# B&R Automation Studio project 8238 (part 16)

```iecst
										_dim1 := MAX(1, _getContainerParamNum.wDimension[1]);
										_dim2 := MAX(1, _getContainerParamNum.wDimension[2]);
										_dim3 := MAX(1, _getContainerParamNum.wDimension[3]);
										_dim4 := MAX(1, _getContainerParamNum.wDimension[4]);

										FOR _i1 := _getContainerParamNum.wMinBound[1] TO _getContainerParamNum.wMinBound[1] + _dim1-1 DO

											FOR _i2 := _getContainerParamNum.wMinBound[2] TO _getContainerParamNum.wMinBound[2] + _dim2 -1 DO

												FOR _i3 := _getContainerParamNum.wMinBound[3] TO _getContainerParamNum.wMinBound[3] + _dim3 -1 DO

													FOR _i4 := _getContainerParamNum.wMinBound[4] TO _getContainerParamNum.wMinBound[4] + _dim4 -1 DO

														IF _wIdxCsvNum <= _PmIntern.CSVDataObjects.MaxIndex.lCSVNum THEN

															_pDoContainerNum.CsvNum[_wIdxCsvNum].wIdxNumPar := _i;
															_pDoContainerNum.CsvNum[_wIdxCsvNum].bRowType := _pDoParamNum.ParamNum[_i].bRowType;
															_pDoContainerNum.CsvNum[_wIdxCsvNum].diValue := _pDoParamNum.ParamNum[_i].diDefValue;

															IF _getContainerParamNum.wCountArray >= 1 THEN

																_pDoContainerNum.CsvNum[_wIdxCsvNum].wArrIdx1 := _i1;

																IF _getContainerParamNum.wCountArray >= 2 THEN

																	_pDoContainerNum.CsvNum[_wIdxCsvNum].wArrIdx2 := _i2;

																	IF _getContainerParamNum.wCountArray >= 3 THEN

																		_pDoContainerNum.CsvNum[_wIdxCsvNum].wArrIdx3 := _i3;

																		IF _getContainerParamNum.wCountArray = 4 THEN

																			_pDoContainerNum.CsvNum[_wIdxCsvNum].wArrIdx4 := _i4;

																		END_IF

																	END_IF

																END_IF

															END_IF

															_wIdxCsvNum := _wIdxCsvNum + 1;

														END_IF

													END_FOR

												END_FOR

											END_FOR

										END_FOR

									END_IF

								END_FOR

								//****************************************************************************************************************
								// Datenobjekte beschreiben (STRING)
								//****************************************************************************************************************
								_wIdxCsvString := 1;

								FOR _i := 1 TO UDINT_TO_UINT(_PmIntern.DataObjects.MaxIndex.lParamString) DO

									_getContainerParamString(enable := TRUE, pLogicStructs := ADR(_pDoLogicalStruct.LogicalStruct[1]), wMaxIdxLogicStructs := UDINT_TO_UINT(_PmIntern.DataObjects.MaxIndex.lLogicalStruct), pParamString := ADR(_pDoParamString.ParamString[_i]));

									IF _getContainerParamString.status = ERR_OK AND _getContainerParamString.iContainer = _pDoContainer.Container[_c].siContainerID THEN

										_dim1 := MAX(1, _getContainerParamString.wDimension[1]);
										_dim2 := MAX(1, _getContainerParamString.wDimension[2]);
										_dim3 := MAX(1, _getContainerParamString.wDimension[3]);
										_dim4 := MAX(1, _getContainerParamString.wDimension[4]);

										FOR _i1 := _getContainerParamString.wMinBound[1] TO _getContainerParamString.wMinBound[1] + _dim1 - 1 DO

											FOR _i2 := _getContainerParamString.wMinBound[2] TO _getContainerParamString.wMinBound[2] + _dim2 - 1 DO

												FOR _i3 := _getContainerParamString.wMinBound[3] TO _getContainerParamString.wMinBound[3] + _dim3 - 1 DO

													FOR _i4 := _getContainerParamString.wMinBound[4] TO _getContainerParamString.wMinBound[4] + _dim4 - 1 DO

														IF _wIdxCsvString <= _PmIntern.CSVDataObjects.MaxIndex.lCSVString THEN

															_pDoContainerString.CsvString[_wIdxCsvString].wIdxStringPar := _i;
															brwcsncpy(ADR(_pDoContainerString.CsvString[_wIdxCsvString].utfValue), ADR(_pDoParamString.ParamString[_i].utfDefValue), 31);

															IF _getContainerParamString.wCountArray >= 1 THEN

																_pDoContainerString.CsvString[_wIdxCsvString].wArrIdx1 := _i1;

																IF _getContainerParamString.wCountArray >= 2 THEN

																	_pDoContainerString.CsvString[_wIdxCsvString].wArrIdx2 := _i2;

																	IF _getContainerParamString.wCountArray >= 3 THEN

																		_pDoContainerString.CsvString[_wIdxCsvString].wArrIdx3 := _i3;

																		IF _getContainerParamString.wCountArray = 4 THEN

																			_pDoContainerString.CsvString[_wIdxCsvString].wArrIdx4 := _i4;

																		END_IF

																	END_IF

																END_IF

															END_IF

															_wIdxCsvString := _wIdxCsvString + 1;

														END_IF

													END_FOR

												END_FOR

											END_FOR

										END_FOR

									END_IF

								END_FOR

								//****************************************************************************************************************
								// Datenobjekte anlegen
								//****************************************************************************************************************

								_dcCSVNum(enable := TRUE, grp := 0, pName := ADR(_PmIntern.ActContainer.sDoNameNum), len := _PmIntern.CSVDataObjects.Size.lCSVNum, MemType := doUSRROM, Option := 0, pCpyData := _PmIntern.CSVDataObjects.TempAdresses.lCSVNum);

								IF (_dcCSVNum.status = ERR_OK) THEN
									_PmIntern.CSVDataObjects.Idents.lCSVNum := _dcCSVNum.ident;
									_PmIntern.CSVDataObjects.Adress.lCSVNum := _dcCSVNum.pDatObjMem;
									_PmIntern.CSVDataObjects.Size.lCSVNum := _dcCSVNum.len;

									_pDoContainerNum ACCESS _PmIntern.CSVDataObjects.Adress.lCSVNum;

									// Es muss auch eine CSV-Datei geschrieben werden
									_PmIntern.xExportContainerCsv := TRUE;

								ELSE

									_PmIntern.Logger.logLevel 	:= arlogLEVEL_INFO;
									_PmIntern.Logger.text		:= 'Create Data Object Numeric failed: Index = {##AttrVar1}. Status: {##AttrVar2}';
									_PmIntern.Logger.var1		:= _PmIntern.ActContainer.siContainerID;
									_PmIntern.Logger.var2		:= _dcCSVNum.status;
									_PmIntern.Logger();

								END_IF

								_dcCSVString(enable := TRUE, grp := 0, pName := ADR(_PmIntern.ActContainer.sDoNameString), len := _PmIntern.CSVDataObjects.Size.lCSVString, MemType := doUSRROM, Option := 0, pCpyData :=_PmIntern.CSVDataObjects.TempAdresses.lCSVString);

								IF (_dcCSVString.status = ERR_OK) THEN
									_PmIntern.CSVDataObjects.Idents.lCSVString := _dcCSVString.ident;
									_PmIntern.CSVDataObjects.Adress.lCSVString := _dcCSVString.pDatObjMem;
									_PmIntern.CSVDataObjects.Size.lCSVString := _dcCSVString.len;

									_pDoContainerString ACCESS _PmIntern.CSVDataObjects.Adress.lCSVString;

									// Es muss auch eine CSV-Datei geschrieben werden
									_PmIntern.xExportContainerCsv := TRUE;

								ELSE

									_PmIntern.Logger.logLevel 	:= arlogLEVEL_INFO;
									_PmIntern.Logger.text		:= 'Create Data Object String failed: Index = {##AttrVar1}. Status: {##AttrVar2}';
									_PmIntern.Logger.var1		:= _PmIntern.ActContainer.siContainerID;
									_PmIntern.Logger.var2		:= _dcCSVString.status;
									_PmIntern.Logger();

								END_IF

								_MemPartFree(enable := TRUE, ident := _MemPartCreate.ident, mem := _PmIntern.CSVDataObjects.TempAdresses.lCSVNum);
								_PmIntern.CSVDataObjects.TempAdresses.lCSVNum := 0;

								_MemPartFree(enable := TRUE, ident := _MemPartCreate.ident, mem := _PmIntern.CSVDataObjects.TempAdresses.lCSVString);
								_PmIntern.CSVDataObjects.TempAdresses.lCSVString := 0;

							ELSE

								_PmIntern.Logger.logLevel 	:= arlogLEVEL_INFO;
								_PmIntern.Logger.text		:= 'MemPartAlloc for Data Object String: Index = {##AttrVar1}. Status: {##AttrVar2}';
								_PmIntern.Logger.var1		:= _PmIntern.ActContainer.siContainerID;
								_PmIntern.Logger.var2		:= _MemPartAlloc.status;
								_PmIntern.Logger();

							END_IF //IF _MemPartAlloc.status = ERR_OK

						ELSE

							_PmIntern.Logger.logLevel 	:= arlogLEVEL_INFO;
							_PmIntern.Logger.text		:= 'MemPartAlloc for Data Object Numeric: Index = {##AttrVar1}. Status: {##AttrVar2}';
							_PmIntern.Logger.var1		:= _PmIntern.ActContainer.siContainerID;
							_PmIntern.Logger.var2		:= _MemPartAlloc.status;
							_PmIntern.Logger();

						END_IF

					END_IF // Direkte Parametrierung

				END_IF // Müssen Datenobjekte angelegt werden

				// Wenn SINGLEmnParam definiert ist, dann wartet die Ausführung hier solange, bis _lSingleStep > _pl_InitState gesetzt wurde
				#ifdef SINGLEmnParam
				REPEAT
		UNTIL
					(_lSingleStep > _pl_InitState) AND (_lLoop >= _lLoopCount) OR NOT _xSingleStep
				END_REPEAT
#endif

				//****************************************************************************************************************
				// CSV-Datei auf Datum prüfen und ggf. einlesen
				//****************************************************************************************************************

				_PmIntern.enInitState := is_TestFileDate;

				// Wenn Datei gefunden, dann Version und Datum bestimmen

				IF _PmIntern.Parse.lFileAdress <> 0   THEN

					brsmemset(_PmIntern.Parse.lLineTableAdress, 0, MNPARAM_MAXPARSELINES * SIZEOF(UDINT));
					brsmemset(_PmIntern.Parse.lLineTableLen, 0, MNPARAM_MAXPARSELINES * SIZEOF(UINT));

					_CountLines.enable 	:= TRUE;
					_CountLines.pFile 		:= _PmIntern.Parse.lFileAdress;
					_CountLines.FileSize 	:= _PmIntern.Parse.lFileSize;
					_CountLines.MaxLines	:= MNPARAM_MAXPARSELINES;
					_CountLines.pAdresses	:= _PmIntern.Parse.lLineTableAdress;
					_CountLines.pLens		:= _PmIntern.Parse.lLineTableLen;

					_CountLines();

					IF _CountLines.status = ERR_OK THEN

						_PmIntern.Parse.lCntLines := _CountLines.CntLines;

						// Suche Versionszeile

						_wStartLine := 1;
						_xFoundVersion := FALSE;
						_xFoundDate := FALSE;
						_xFoundMachineNo := FALSE;

						REPEAT

							_GetCsvDat.enable := TRUE;
							brwcsncpy( ADR(_GetCsvDat.utfCsvString), _plLineAdress[_wStartLine], MIN(299, _pwLineLen[_wStartLine]));
							_GetCsvDat();
							IF _GetCsvDat.RowType = MNPARAM_CSV_HEADER_VERSION THEN

								_CsvHeaderVersion := _GetCsvDat.HeaderVersion;
								_xFoundVersion := TRUE;

							ELSIF _GetCsvDat.RowType = MNPARAM_CSV_HEADER_TIMESTAMP THEN

								_CsvHeaderDate := _GetCsvDat.HeaderTime;
								_xFoundDate := TRUE;

							ELSIF _GetCsvDat.RowType = MNPARAM_CSV_HEADER_MACHINENO THEN

								_CsvHeaderMachineNo := _GetCsvDat.HeaderMachineNo;
								_xFoundMachineNo := TRUE;

							END_IF

							_wStartLine := _wStartLine + 1;

						UNTIL
							(_xFoundDate AND _xFoundVersion AND _xFoundMachineNo) OR _wStartLine > _PmIntern.Parse.lCntLines
						END_REPEAT

						_PmIntern.ActContainer.xDataImported := FALSE;

						IF _xFoundDate AND _xFoundVersion AND _xFoundMachineNo THEN

							// Ist der Maschinentyp OK ?
							IF brwcscmp(ADR(_CsvHeaderVersion.utfMachineType),ADR(_pDoContainer.Header.Version.utfMachineType)) = 0 THEN

								// Ist die Maschinennummer OK ?
								IF brwcscmp(ADR(_CsvHeaderMachineNo.utfMachineNo),ADR(IFmnParam.Out.utfMachineNumber)) = 0 THEN

									// Ist die CSV-Datei neuer als die Daten in den DO ?
									IF _pDoContainerNum.Header.Time.dtTimestamp < _CsvHeaderDate.dtTimestamp THEN

										//****************************************************************************************************************
										// Datenobjekte für das Importieren in den Hauptspeicher kopieren
										//****************************************************************************************************************

										_PmIntern.enInitState := is_ImportData1;

										//##20110901AH
										_PmIntern.Logger.logLevel 	:= arlogLEVEL_INFO;
										_PmIntern.Logger.text		:= 'Import Container Index = {##AttrVar1}. Index: {##AttrVar2}';
										_PmIntern.Logger.var1		:= _PmIntern.ActContainer.siContainerID;
										_PmIntern.Logger.var2		:= _PmIntern.ActContainer.wIndexIndirect;
										_PmIntern.Logger();

										// Numerische Daten
										_diCSVNum(enable := TRUE, pName := ADR(_PmIntern.ActContainer.sDoNameNum));

										IF _diCSVNum.status = ERR_OK THEN

											_PmIntern.CSVDataObjects.Idents.lCSVNum := _diCSVNum.ident;
											_PmIntern.CSVDataObjects.Adress.lCSVNum := _diCSVNum.pDatObjMem;
											_PmIntern.CSVDataObjects.Size.lCSVNum := _diCSVNum.len;

											_MemPartAlloc(enable :=TRUE, ident := _MemPartCreate.ident, len := _diCSVNum.len);

											IF _MemPartAlloc.status = ERR_OK THEN

												_drCSVNum(enable := TRUE, ident := _diCSVNum.ident, Offset := 0, pDestination := _MemPartAlloc.mem, len := _MemPartAlloc.len);

												IF _drCSVNum.status = ERR_OK THEN

													// Im Hauptspeicher ist wieder Schreibzugriff möglich
													_PmIntern.CSVDataObjects.TempAdresses.lCSVNum := _MemPartAlloc.mem;
													_pDoContainerNum ACCESS _PmIntern.CSVDataObjects.TempAdresses.lCSVNum;

													// Maximalen Index für Einträge prüfen. Lücken sollte es nicht geben
													_PmIntern.CSVDataObjects.MaxIndex.lCSVNum := ( (_pDoContainerNum.Header.Do.lActEndPos - SIZEOF(mnParam_CsvDynHeader_typ)) / SIZEOF(_pDoContainerNum.CsvNum[1]) );

												ELSE

													_PmIntern.CSVDataObjects.Idents.lCSVNum := 0;
													_PmIntern.CSVDataObjects.Adress.lCSVNum := 0;
													_PmIntern.CSVDataObjects.Size.lCSVNum := 0;

													_MemPartFree(enable := TRUE, ident := _MemPartCreate.ident, mem := _MemPartAlloc.mem);

													_PmIntern.Logger.logLevel 	:= arlogLEVEL_INFO;
													_PmIntern.Logger.text		:= 'Read Data Object Numeric Container: Index = {##AttrVar1}. Status: {##AttrVar2}';
													_PmIntern.Logger.var1		:= _PmIntern.ActContainer.siContainerID;
													_PmIntern.Logger.var2		:= _drCSVNum.status;
													_PmIntern.Logger();

												END_IF

											ELSE

												_PmIntern.CSVDataObjects.Idents.lCSVNum := 0;
												_PmIntern.CSVDataObjects.Adress.lCSVNum := 0;
												_PmIntern.CSVDataObjects.Size.lCSVNum := 0;

												_PmIntern.Logger.logLevel 	:= arlogLEVEL_INFO;
												_PmIntern.Logger.text		:= 'MemPartAlloc for Read Data Object Numeric Container: Index = {##AttrVar1}. Status: {##AttrVar2}';
												_PmIntern.Logger.var1		:= _PmIntern.ActContainer.siContainerID;
												_PmIntern.Logger.var2		:= _MemPartAlloc.status;
												_PmIntern.Logger();

											END_IF // _MemPartAlloc.status

										ELSE

											_PmIntern.Logger.logLevel 	:= arlogLEVEL_INFO;
											_PmIntern.Logger.text		:= 'Data Object Numeric Container does not exist: Index = {##AttrVar1}. Status: {##AttrVar2}';
											_PmIntern.Logger.var1		:= _PmIntern.ActContainer.siContainerID;
											_PmIntern.Logger.var2		:= _diCSVNum.status;
											_PmIntern.Logger();

										END_IF // _diCSVNum.status

										// String Daten
										_diCSVString(enable := TRUE, pName := ADR(_PmIntern.ActContainer.sDoNameString));

										IF _diCSVString.status = ERR_OK THEN

											_PmIntern.CSVDataObjects.Idents.lCSVString := _diCSVString.ident;
											_PmIntern.CSVDataObjects.Adress.lCSVString := _diCSVString.pDatObjMem;
											_PmIntern.CSVDataObjects.Size.lCSVString := _diCSVString.len;

											_MemPartAlloc(enable :=TRUE, ident := _MemPartCreate.ident, len := _diCSVString.len);

											IF _MemPartAlloc.status = ERR_OK THEN

												_drCSVString(enable := TRUE, ident := _diCSVString.ident, Offset := 0, pDestination := _MemPartAlloc.mem, len := _MemPartAlloc.len);

												IF _drCSVString.status = ERR_OK THEN

													// Im Hauptspeicher ist wieder Schreibzugriff möglich
													_PmIntern.CSVDataObjects.TempAdresses.lCSVString := _MemPartAlloc.mem;
													_pDoContainerString ACCESS _PmIntern.CSVDataObjects.TempAdresses.lCSVString;

													// Maximalen Index für Einträge prüfen. Lücken sollte es nicht geben
													_PmIntern.CSVDataObjects.MaxIndex.lCSVString := ( (_pDoContainerString.Header.Do.lActEndPos - SIZEOF(mnParam_CsvDynHeader_typ)) / SIZEOF(_pDoContainerString.CsvString[1]) );

												ELSE

													_PmIntern.CSVDataObjects.Idents.lCSVString := 0;
													_PmIntern.CSVDataObjects.Adress.lCSVString := 0;
													_PmIntern.CSVDataObjects.Size.lCSVString := 0;

													_MemPartFree(enable := TRUE, ident := _MemPartCreate.ident, mem := _MemPartAlloc.mem);

													_PmIntern.Logger.logLevel 	:= arlogLEVEL_INFO;
													_PmIntern.Logger.text		:= 'Read Data Object String Container: Index = {##AttrVar1}. Status: {##AttrVar2}';
													_PmIntern.Logger.var1		:= _PmIntern.ActContainer.siContainerID;
													_PmIntern.Logger.var2		:= _drCSVString.status;
													_PmIntern.Logger();

												END_IF

											ELSE

												_PmIntern.Logger.logLevel 	:= arlogLEVEL_INFO;
												_PmIntern.Logger.text		:= 'MemPartAlloc for Read Data Object String Container: Index = {##AttrVar1}. Status: {##AttrVar2}';
												_PmIntern.Logger.var1		:= _PmIntern.ActContainer.siContainerID;
												_PmIntern.Logger.var2		:= _MemPartAlloc.status;
												_PmIntern.Logger();

											END_IF // _MemPartAlloc.status

										ELSE

											_PmIntern.Logger.logLevel 	:= arlogLEVEL_INFO;
											_PmIntern.Logger.text		:= 'Data Object String Container does not exist: Index = {##AttrVar1}. Status: {##AttrVar2}';
											_PmIntern.Logger.var1		:= _PmIntern.ActContainer.siContainerID;
											_PmIntern.Logger.var2		:= _diCSVString.status;
											_PmIntern.Logger();

										END_IF // _diCSVNum.status

										// Wenn SINGLEmnParam definiert ist, dann wartet die Ausführung hier solange, bis _lSingleStep > _pl_InitState gesetzt wurde
										#ifdef SINGLEmnParam
										REPEAT
											UNTIL
											_lSingleStep > _pl_InitState OR NOT _xSingleStep
										END_REPEAT
										#endif

										//****************************************************************************************************************
										// Alles auf Default setzen
										//****************************************************************************************************************

										FOR _i := 1 TO UDINT_TO_UINT(_PmIntern.CSVDataObjects.MaxIndex.lCSVNum) DO

											IF _pDoContainerNum.CsvNum[_i].wIdxNumPar > 0 AND _pDoContainerNum.CsvNum[_i].wIdxNumPar <= _PmIntern.ActContainer.lCountParamNum THEN

												_pDoContainerNum.CsvNum[_i].diValue := _pDoParamNum.ParamNum[_pDoContainerNum.CsvNum[_i].wIdxNumPar].diDefValue;
												_pDoContainerNum.CsvNum[_i].xChanged := FALSE;

											END_IF

										END_FOR

										FOR _i := 1 TO UDINT_TO_UINT(_PmIntern.CSVDataObjects.MaxIndex.lCSVString) DO

											IF _pDoContainerString.CsvString[_i].wIdxStringPar > 0 AND _pDoContainerString.CsvString[_i].wIdxStringPar <= _PmIntern.ActContainer.lCountParamString THEN

												_pDoContainerString.CsvString[_i].utfValue := _pDoParamString.ParamString[_pDoContainerString.CsvString[_i].wIdxStringPar].utfDefValue;
												_pDoContainerString.CsvString[_i].xChanged := FALSE;

											END_IF

										END_FOR

										//****************************************************************************************************************
										// CSV-Datei importieren
										//****************************************************************************************************************

										_PmIntern.enInitState := is_ImportData2;

										_binarySearchNum.enable := TRUE;
										_binarySearchNum.lpList := _PmIntern.CSVDataObjects.TempAdresses.lCSVNum;
										_binarySearchNum.lMaxRow := _PmIntern.CSVDataObjects.MaxIndex.lCSVNum;

										_binarySearchString.enable := TRUE;
										_binarySearchString.lpList := _PmIntern.CSVDataObjects.TempAdresses.lCSVString;
										_binarySearchString.lMaxRow := _PmIntern.CSVDataObjects.MaxIndex.lCSVString;

										REPEAT

											_GetCsvDat.enable := TRUE;
											brwcsncpy( ADR(_GetCsvDat.utfCsvString), _plLineAdress[_wStartLine], MIN(299, _pwLineLen[_wStartLine]));
											_GetCsvDat();

											IF _GetCsvDat.RowType = 10 OR _GetCsvDat.RowType = 11 THEN

												_binarySearchNum.CsvStructNum := _GetCsvDat.CsvNumRow;
												_binarySearchNum();

												IF _binarySearchNum.status = 0 THEN

													_pDoContainerNum.CsvNum[_binarySearchNum.lFoundRow] := _GetCsvDat.CsvNumRow;

													_LP(pCsvNumRow := ADR(_pDoContainerNum.CsvNum[_binarySearchNum.lFoundRow]), pParamNum := ADR(_pDoParamNum.ParamNum[_GetCsvDat.CsvNumRow.wIdxNumPar]) );

													_pDoContainerNum.CsvNum[_binarySearchNum.lFoundRow].xChanged := _pDoParamNum.ParamNum[_GetCsvDat.CsvNumRow.wIdxNumPar].diDefValue <> _GetCsvDat.CsvNumRow.diValue;

												ELSE

													_PmIntern.Logger.logLevel 	:= arlogLEVEL_INFO;
													_PmIntern.Logger.text		:= 'Binary Search Numeric. Container Index = {##AttrVar1}. Status: {##AttrVar2}: ';
													brsitoa(_GetCsvDat.CsvNumRow.wIdxNumPar, ADR(_sNumeric));
													_PmIntern.Logger.text		:= CONCAT(_PmIntern.Logger.text, _sNumeric);
													_PmIntern.Logger.text		:= CONCAT(_PmIntern.Logger.text, ', ');
													brsitoa(_GetCsvDat.CsvNumRow.wArrIdx1, ADR(_sNumeric));
													_PmIntern.Logger.text		:= CONCAT(_PmIntern.Logger.text, _sNumeric);
													_PmIntern.Logger.text		:= CONCAT(_PmIntern.Logger.text, ', ');
													brsitoa(_GetCsvDat.CsvNumRow.wArrIdx2, ADR(_sNumeric));
													_PmIntern.Logger.text		:= CONCAT(_PmIntern.Logger.text, _sNumeric);
													_PmIntern.Logger.text		:= CONCAT(_PmIntern.Logger.text, ', ');
													brsitoa(_GetCsvDat.CsvNumRow.wArrIdx3, ADR(_sNumeric));
													_PmIntern.Logger.text		:= CONCAT(_PmIntern.Logger.text, _sNumeric);
													_PmIntern.Logger.text		:= CONCAT(_PmIntern.Logger.text, ', ');
													brsitoa(_GetCsvDat.CsvNumRow.wArrIdx4, ADR(_sNumeric));
													_PmIntern.Logger.text		:= CONCAT(_PmIntern.Logger.text, _sNumeric);
													_PmIntern.Logger.var1		:= _PmIntern.ActContainer.siContainerID;
													_PmIntern.Logger.var2		:= _binarySearchNum.status;
													_PmIntern.Logger();

												END_IF

											ELSIF _GetCsvDat.RowType = 20 THEN

												_binarySearchString.CsvStructString := _GetCsvDat.CsvStringRow;
												_binarySearchString();

												IF _binarySearchString.status = 0 THEN

													_pDoContainerString.CsvString[_binarySearchString.lFoundRow] := _GetCsvDat.CsvStringRow;

													_pDoContainerString.CsvString[_binarySearchString.lFoundRow].xChanged := brwcscmp(ADR(_pDoParamString.ParamString[_GetCsvDat.CsvStringRow.wIdxStringPar].utfDefValue), ADR(_GetCsvDat.CsvStringRow.utfValue)) <> 0;

												ELSE

													_PmIntern.Logger.logLevel 	:= arlogLEVEL_INFO;
													_PmIntern.Logger.text		:= 'Binary Search String. Container Index = {##AttrVar1}. Status: {##AttrVar2}: ';
													brsitoa(_GetCsvDat.CsvStringRow.wIdxStringPar, ADR(_sNumeric));
													_PmIntern.Logger.text		:= CONCAT(_PmIntern.Logger.text, _sNumeric);
													_PmIntern.Logger.text		:= CONCAT(_PmIntern.Logger.text, ', ');
													brsitoa(_GetCsvDat.CsvStringRow.wArrIdx1, ADR(_sNumeric));
													_PmIntern.Logger.text		:= CONCAT(_PmIntern.Logger.text, _sNumeric);
													_PmIntern.Logger.text		:= CONCAT(_PmIntern.Logger.text, ', ');
													brsitoa(_GetCsvDat.CsvStringRow.wArrIdx2, ADR(_sNumeric));
													_PmIntern.Logger.text		:= CONCAT(_PmIntern.Logger.text, _sNumeric);
													_PmIntern.Logger.text		:= CONCAT(_PmIntern.Logger.text, ', ');
													brsitoa(_GetCsvDat.CsvStringRow.wArrIdx3, ADR(_sNumeric));
													_PmIntern.Logger.text		:= CONCAT(_PmIntern.Logger.text, _sNumeric);
													_PmIntern.Logger.text		:= CONCAT(_PmIntern.Logger.text, ', ');
													brsitoa(_GetCsvDat.CsvStringRow.wArrIdx4, ADR(_sNumeric));
													_PmIntern.Logger.text		:= CONCAT(_PmIntern.Logger.text, _sNumeric);
													_PmIntern.Logger.var1		:= _PmIntern.ActContainer.siContainerID;
													_PmIntern.Logger.var2		:= _binarySearchString.status;
													_PmIntern.Logger();

												END_IF

											END_IF

											_wStartLine := _wStartLine + 1;

											UNTIL
											_wStartLine > _PmIntern.Parse.lCntLines
										END_REPEAT

										// Wenn SINGLEmnParam definiert ist, dann wartet die Ausführung hier solange, bis _lSingleStep > _pl_InitState gesetzt wurde
										#ifdef SINGLEmnParam
										REPEAT
											UNTIL
											_lSingleStep > _pl_InitState OR NOT _xSingleStep
										END_REPEAT
										#endif

										//****************************************************************************************************************
										// DO schreiben
										//****************************************************************************************************************

										_PmIntern.enInitState := is_ImportData3;

										_DTGetTime(enable := TRUE);
										_pDoContainerNum.Header.Time.dtTimestamp := _DTGetTime.DT1;
										_pDoContainerString.Header.Time.dtTimestamp := _DTGetTime.DT1;

										_pDoContainerNum.Header.Container.xWriteProtected := _PmIntern.ActContainer.xWriteProtected;
										_pDoContainerString.Header.Container.xWriteProtected := _PmIntern.ActContainer.xWriteProtected;

										IF _PmIntern.CSVDataObjects.Idents.lCSVNum <> 0 THEN

											_dwCSVNum(enable := TRUE, ident := _PmIntern.CSVDataObjects.Idents.lCSVNum, Offset := 0, pSource := _PmIntern.CSVDataObjects.TempAdresses.lCSVNum, len := _PmIntern.CSVDataObjects.Size.lCSVNum);

											IF _dwCSVNum.status <> ERR_OK THEN

												_PmIntern.Logger.logLevel 	:= arlogLEVEL_INFO;
												_PmIntern.Logger.text		:= 'Write Data Object Numeric Container: Index = {##AttrVar1}. Status: {##AttrVar2}';
												_PmIntern.Logger.var1		:= _PmIntern.ActContainer.siContainerID;
												_PmIntern.Logger.var2		:= _dwCSVNum.status;
												_PmIntern.Logger();

											END_IF

											_MemPartFree(enable := TRUE, ident  := _MemPartCreate.ident, mem := _PmIntern.CSVDataObjects.TempAdresses.lCSVNum);

											_pDoContainerNum ACCESS _PmIntern.CSVDataObjects.Adress.lCSVNum;

											_PmIntern.CSVDataObjects.TempAdresses.lCSVNum := 0;

										END_IF

										IF _PmIntern.CSVDataObjects.Idents.lCSVString <> 0 THEN

											_dwCSVString(enable := TRUE, ident := _PmIntern.CSVDataObjects.Idents.lCSVString, Offset := 0, pSource := _PmIntern.CSVDataObjects.TempAdresses.lCSVString, len := _PmIntern.CSVDataObjects.Size.lCSVString);

											IF _dwCSVString.status <> ERR_OK THEN

												_PmIntern.Logger.logLevel 	:= arlogLEVEL_INFO;
												_PmIntern.Logger.text		:= 'Write Data Object String Container: Index = {##AttrVar1}. Status: {##AttrVar2}';
												_PmIntern.Logger.var1		:= _PmIntern.ActContainer.siContainerID;
												_PmIntern.Logger.var2		:= _dwCSVString.status;
												_PmIntern.Logger();

											END_IF

											_MemPartFree(enable := TRUE, ident  := _MemPartCreate.ident, mem := _PmIntern.CSVDataObjects.TempAdresses.lCSVString);

											_pDoContainerString ACCESS _PmIntern.CSVDataObjects.Adress.lCSVString;

											_PmIntern.CSVDataObjects.TempAdresses.lCSVString := 0;

										END_IF

										_PmIntern.ActContainer.xDataImported := TRUE;

									ELSIF _pDoContainerNum.Header.Time.dtTimestamp > _CsvHeaderDate.dtTimestamp THEN

										_PmIntern.ActContainer.xDataImported := TRUE;

									END_IF

								ELSE

									//Ungültige Maschinennummer
									_PmIntern.Logger.logLevel 	:= arlogLEVEL_INFO;
									_PmIntern.Logger.text		:= 'Wrong Machineno. in CSV-Container: Index = {##AttrVar1}/{##AttrVar2}. ';
									_PmIntern.Logger.var1		:= _PmIntern.ActContainer.siContainerID;
									_PmIntern.Logger.var2		:= _PmIntern.ActContainer.wIndexIndirect;
									_PmIntern.Logger();

								END_IF

							ELSE

								//Ungültige Datei
								_PmIntern.Logger.logLevel 	:= arlogLEVEL_INFO;
								_PmIntern.Logger.text		:= 'Wrong Machine Type in CSV-Container: Index = {##AttrVar1}/{##AttrVar2}. ';
								_PmIntern.Logger.var1		:= _PmIntern.ActContainer.siContainerID;
								_PmIntern.Logger.var2		:= _PmIntern.ActContainer.wIndexIndirect;
								_PmIntern.Logger();

							END_IF

						ELSE

							//Ungültige Datei
							_PmIntern.Logger.logLevel 	:= arlogLEVEL_INFO;
							_PmIntern.Logger.text		:= 'No Version, date or machineno. in CSV-Container: Index = {##AttrVar1}/{##AttrVar2}. ';
							_PmIntern.Logger.var1		:= _PmIntern.ActContainer.siContainerID;
							_PmIntern.Logger.var2		:= _PmIntern.ActContainer.wIndexIndirect;
							_PmIntern.Logger();

						END_IF

					ELSE

						//Ungültige Datei
						_PmIntern.Logger.logLevel 	:= arlogLEVEL_INFO;
						_PmIntern.Logger.text		:= 'Fault in Counting Lines of CSV-Container: Index = {##AttrVar1}. Status: {##AttrVar2}';
						_PmIntern.Logger.var1		:= _PmIntern.ActContainer.siContainerID;
						_PmIntern.Logger.var2		:= _CountLines.status;
						_PmIntern.Logger();

					END_IF

					// Temporären Speicher zum Parsen der csv-Datei wieder frei geben
					_MemPartFree(enable := TRUE, ident  := _MemPartCreate.ident, mem := _PmIntern.Parse.lFileAdress);
					_PmIntern.Parse.lFileAdress := 0;

				END_IF

				// Wenn SINGLEmnParam definiert ist, dann wartet die Ausführung hier solange, bis _lSingleStep > _pl_InitState gesetzt wurde
#ifdef SINGLEmnParam
				REPEAT
					UNTIL
					(_lSingleStep > _pl_InitState) AND (_lLoop >= _lLoopCount) OR NOT _xSingleStep
				END_REPEAT
#endif

				//****************************************************************************************************************
				// Datenobjekt für indirekte Parametrierung identifizieren
				//****************************************************************************************************************

				_PmIntern.enInitState := is_SetValue1;

				// Bei indirekter Parametrierung, das Binär-Datenobjekt
				IF _PmIntern.ActContainer.bDirect = 0 AND (_PmIntern.CSVDataObjects.MaxIndex.lCSVNum > 0 OR _PmIntern.CSVDataObjects.MaxIndex.lCSVString > 0) AND _PmIntern.ActContainer.xDataImported THEN

					_diDO(enable := TRUE, pName := ADR(_PmIntern.ActContainer.sDoName));

					IF _diDO.status = ERR_OK THEN

						_PmIntern.CSVDataObjects.Idents.lDataObjekt := _diDO.ident;

						_wStatus := PV_xgetadr(ADR(_PmIntern.ActContainer.sStrucRoot), ADR(_PmIntern.CSVDataObjects.TempAdresses.lDataObjekt), ADR(_PmIntern.CSVDataObjects.Size.lDataObjekt));

						IF _wStatus = ERR_OK THEN

							_drDO(enable := TRUE, ident := _diDO.ident, Offset := 0, pDestination := _PmIntern.CSVDataObjects.TempAdresses.lDataObjekt, len := _PmIntern.CSVDataObjects.Size.lDataObjekt);

							IF _drDO.status <> ERR_OK THEN

								//Ungültige Datei
								_PmIntern.Logger.logLevel 	:= arlogLEVEL_INFO;
								_PmIntern.Logger.text		:= 'Data Object Read Binary Container: Index = {##AttrVar1}. Status: {##AttrVar2}';
								_PmIntern.Logger.var1		:= _PmIntern.ActContainer.siContainerID;
								_PmIntern.Logger.var2		:= _drDO.status;
								_PmIntern.Logger();

							END_IF

						ELSE

							_PmIntern.Logger.logLevel 	:= arlogLEVEL_INFO;
							_PmIntern.Logger.text		:= CONCAT('Root element does not exist: Index = {##AttrVar1}. Status: {##AttrVar2} - ', _PmIntern.ActContainer.sStrucRoot);
							_PmIntern.Logger.var1		:= _PmIntern.ActContainer.siContainerID;
							_PmIntern.Logger.var2		:= _wStatus;
							_PmIntern.Logger();

						END_IF

					ELSE

						_PmIntern.Logger.logLevel 	:= arlogLEVEL_INFO;
						_PmIntern.Logger.text		:= 'Data Object Binary does not exist! Container: Index = {##AttrVar1}. Status: {##AttrVar2}';
						_PmIntern.Logger.var1		:= _PmIntern.ActContainer.siContainerID;
						_PmIntern.Logger.var2		:= _diDO.status;
						_PmIntern.Logger();

					END_IF

				END_IF

				// Wenn SINGLEmnParam definiert ist, dann wartet die Ausführung hier solange, bis _lSingleStep > _pl_InitState gesetzt wurde
				#ifdef SINGLEmnParam
				REPEAT
					UNTIL
					(_lSingleStep > _pl_InitState) AND (_lLoop >= _lLoopCount) OR NOT _xSingleStep
				END_REPEAT
#endif

				//****************************************************************************************************************
				// Daten setzen
				//****************************************************************************************************************

				_PmIntern.enInitState := is_SetValue2;

				IF _PmIntern.ActContainer.bDirect = 1 OR _PmIntern.CSVDataObjects.TempAdresses.lDataObjekt > 0 THEN

					// Numerische Parameter schreiben
					FOR _i := 1 TO UDINT_TO_UINT(_PmIntern.CSVDataObjects.MaxIndex.lCSVNum) DO

						IF _pDoContainerNum.CsvNum[_i].wIdxNumPar > 0 AND _pDoContainerNum.CsvNum[_i].wIdxNumPar <= _PmIntern.DataObjects.MaxIndex.lParamNum THEN

							_PN := _pDoParamNum.ParamNum[_pDoContainerNum.CsvNum[_i].wIdxNumPar];

							_CN := _pDoContainerNum.CsvNum[_i];

							GetArrayPV(pPV := ADR(_PN.sAdresse), pStructRoot := ADR(_PmIntern.ActContainer.sStrucRoot), pPVFilled := ADR(_sPVAdress), idx1 :=_CN.wArrIdx1, idx2:=_CN.wArrIdx2, idx3:=_CN.wArrIdx3, idx4:=_CN.wArrIdx4);

							IF _CN.bRowType = 0 THEN

								_WritePVNum(pAdress := ADR(_sPVAdress), diValue := _CN.diValue);

							ELSE

								_pdiValue ACCESS ADR(_rValue);
								_pdiValue := _CN.diValue;
								_WritePVrNum(pAdress := ADR(_sPVAdress), rValue := _rValue);

							END_IF

							IF _WritePVNum.status <> ERR_OK THEN

								_PmIntern.Logger.logLevel 	:= arlogLEVEL_INFO;
								_PmIntern.Logger.text		:= CONCAT('Write Numeric PV Status {##AttrVar1} - ',_sPVAdress);
								_PmIntern.Logger.var1		:= _WritePVNum.status;
								_PmIntern.Logger.var2		:= 0;
								_PmIntern.Logger();

							END_IF

						ELSE

							_PmIntern.Logger.logLevel 	:= arlogLEVEL_INFO;
							_PmIntern.Logger.text		:= 'Wrong Numeric Parameter Reference : {##AttrVar1}';
							_PmIntern.Logger.var1		:= _pDoContainerNum.CsvNum[_i].wIdxNumPar;
							_PmIntern.Logger.var2		:= 0;
							_PmIntern.Logger();

						END_IF

					END_FOR

					// String Parameter schreiben
					FOR _i := 1 TO UDINT_TO_UINT(_PmIntern.CSVDataObjects.MaxIndex.lCSVString) DO

						IF _pDoContainerString.CsvString[_i].wIdxStringPar > 0 AND _pDoContainerString.CsvString[_i].wIdxStringPar <= _PmIntern.DataObjects.MaxIndex.lParamString THEN

							_PS := _pDoParamString.ParamString[_pDoContainerString.CsvString[_i].wIdxStringPar];

							_CS := _pDoContainerString.CsvString[_i];

							GetArrayPV(pPV := ADR(_PS.sAdresse), pStructRoot := ADR(_PmIntern.ActContainer.sStrucRoot), pPVFilled := ADR(_sPVAdress), idx1 :=_CS.wArrIdx1, idx2:=_CS.wArrIdx2, idx3:=_CS.wArrIdx3, idx4:=_CS.wArrIdx4);

							IF _pDoContainerString.CsvString[_i].wIdxStringPar = MNPARAM_PARIDX_MACHINENAME AND _c = MNPARAM_IDX_MACHINENAMECONTAINER THEN
								mnParamStatAd.utfMachineName := _CS.utfValue;
							END_IF

							_WritePVString(pAdress := ADR(_sPVAdress), p_utfValue := ADR(_CS.utfValue));

							IF _WritePVString.status <> ERR_OK THEN

								_PmIntern.Logger.logLevel 	:= arlogLEVEL_INFO;
								_PmIntern.Logger.text		:= CONCAT('Write String PV Status {##AttrVar1} - ',_sPVAdress);
								_PmIntern.Logger.var1		:= _WritePVString.status;
								_PmIntern.Logger.var2		:= 0;
								_PmIntern.Logger();

							END_IF

						ELSE

							_PmIntern.Logger.logLevel 	:= arlogLEVEL_INFO;
							_PmIntern.Logger.text		:= 'Wrong String Parameter Reference : {##AttrVar1}';
							_PmIntern.Logger.var1		:= _pDoContainerString.CsvString[_i].wIdxStringPar;
							_PmIntern.Logger.var2		:= 0;
							_PmIntern.Logger();

						END_IF

					END_FOR

				END_IF

				//****************************************************************************************************************
				// Datenobjekt für indirekte Parametrierung sichern
				//****************************************************************************************************************

				_PmIntern.enInitState := is_SetValue3;

				IF _PmIntern.ActContainer.bDirect = 0 AND _PmIntern.CSVDataObjects.Idents.lDataObjekt > 0 AND _PmIntern.CSVDataObjects.TempAdresses.lDataObjekt > 0 THEN

					_dwDO(enable := TRUE, ident := _PmIntern.CSVDataObjects.Idents.lDataObjekt, Offset := 0, pSource := _PmIntern.CSVDataObjects.TempAdresses.lDataObjekt, len := _PmIntern.CSVDataObjects.Size.lDataObjekt);

					IF _dwDO.status <> ERR_OK THEN

						_PmIntern.Logger.logLevel 	:= arlogLEVEL_INFO;
						_PmIntern.Logger.text		:= 'Writing Binary Data Object for Container Index: {##AttrVar1}. Status : {##AttrVar2}';
						_PmIntern.Logger.var1		:= _PmIntern.ActContainer.siContainerID;
						_PmIntern.Logger.var2		:= _dwDO.status;
						_PmIntern.Logger();

					END_IF

					_PmIntern.CSVDataObjects.Adress.lDataObjekt := 0;
					_PmIntern.CSVDataObjects.Idents.lDataObjekt := 0;
					_PmIntern.CSVDataObjects.Size.lDataObjekt := 0;
					_PmIntern.CSVDataObjects.TempAdresses.lDataObjekt := 0;

				END_IF

				//****************************************************************************************************************
				// CSV-Dateien in das Export-Verzeichnis schreiben
				//****************************************************************************************************************

				_PmIntern.enInitState := is_ExpCSV;

				IF _PmIntern.xExportContainerCsv OR _PmIntern.ActContainer.xDataImported OR (NOT _PmIntern.xResetConateinerDOs AND NOT _PmIntern.ActContainer.xExportfileExist) THEN

					_PmIntern.ExpSettings.sCfDeviceName := KG_DEVICE_COMPACTFLASH;
					_PmIntern.ExpSettings.sPath := MNPARAM_PATH_EXPORT;
					_PmIntern.ExpSettings.sFilename := _PmIntern.ActContainer.sCsvName;

					_ec(Enable := TRUE, pIntern := ADR(_PmIntern));

					IF _ec.Status = ERR_OK THEN

						_wIdxToc := _PmIntern.TOC.wStartIdx[_PmIntern.ActContainer.siContainerID * (-1)] + _PmIntern.ActContainer.wIndexIndirect - _PmIntern.ActContainer.wMinBound;

						IF _wIdxToc >= 1 AND _wIdxToc <= MNPARAM_CNT_CSVFILES THEN

							_PmIntern.TOC.TocEntry[_wIdxToc].xExist := TRUE;
							_PmIntern.TOC.TocEntry[_wIdxToc].iContainerID := _PmIntern.ActContainer.siContainerID;
							IF _PmIntern.ActContainer.bDirect = 1 THEN
								_PmIntern.TOC.TocEntry[_wIdxToc].wInstance := 0;
							ELSE
								_PmIntern.TOC.TocEntry[_wIdxToc].wInstance := _PmIntern.ActContainer.wIndexIndirect;
							END_IF
							_PmIntern.TOC.TocEntry[_wIdxToc].dtTimestamp :=  _pDoContainerNum.Header.Time.dtTimestamp;

						END_IF

					ELSE

						_PmIntern.Logger.logLevel 	:= arlogLEVEL_INFO;
						_PmIntern.Logger.text		:= 'Writing CSV for Container Index: {##AttrVar1}. Status : {##AttrVar2}';
						_PmIntern.Logger.var1		:= _PmIntern.ActContainer.siContainerID;
						_PmIntern.Logger.var2		:= _ec.Status;
						_PmIntern.Logger();

					END_IF

				END_IF

				// Wenn SINGLEmnParam definiert ist, dann wartet die Ausführung hier solange, bis _lSingleStep > _pl_InitState gesetzt wurde
				#ifdef SINGLEmnParam
				REPEAT
					UNTIL
					(_lSingleStep > _pl_InitState) AND (_lLoop >= _lLoopCount) OR NOT _xSingleStep
				END_REPEAT
				#endif

				//****************************************************************************************************************
				// Nächste Iteration
				//****************************************************************************************************************

				// Bei indirekter Parametrierung mit Instanzen, die nächste Instanz wählen
				IF _PmIntern.ActContainer.bDirect = 0 AND _PmIntern.ActContainer.wDimension > 0 THEN
//					_PmIntern.ActContainer.wIndexIndirect := _PmIntern.ActContainer.wIndexIndirect + 1;
					_wIndexIndirect := _wIndexIndirect + 1;
				END_IF

				_lLoopCount := _lLoopCount + 1;

				UNTIL
				// Direkte Parametrierung, Indirekte Parametrierung ohne Instanzen oder Indirekte Parametrierung und alle Instanzen abgearbeitet
//				_PmIntern.ActContainer.bDirect = 1 OR ( _PmIntern.ActContainer.bDirect = 0 AND _PmIntern.ActContainer.wIndexIndirect >= (_PmIntern.ActContainer.wMinBound + _PmIntern.ActContainer.wDimension)  )
				_PmIntern.ActContainer.bDirect = 1 OR ( _PmIntern.ActContainer.bDirect = 0 AND _wIndexIndirect >= (_PmIntern.ActContainer.wMinBound + _PmIntern.ActContainer.wDimension)  )
			END_REPEAT

		END_FOR	// _c - Über alle Container iterieren

		_PmIntern.ExpSettings.sCfDeviceName := KG_DEVICE_COMPACTFLASH;
		_PmIntern.ExpSettings.sPath := MNPARAM_PATH_EXPORT;

		_ExportTableOfContent(Enable := TRUE, pIntern := ADR(_PmIntern));

		IF _ExportTableOfContent.Status = ERR_OK THEN

			mnParamStatAd.dtExportContent := _ExportTableOfContent.dtTocWritten;

		END_IF

		//=========================================================================================
		//							ENDE DATENCONTAINER PRUEFEN UND EINLESEN
		//=========================================================================================

		IFmnParam.Out.Edit.wIdxContainerNamelist := MNPARAM_IDX_PROGCONTAINER;
		IFmnParam.Out.Edit.wParIdxNamelist := MNPARAM_PARIDX_PROGNAME;

		_actFillNamelist;

		// Initialisierung Fehlerfrei abgeschlossen
		_xInitOk := TRUE;

		UNTIL
		TRUE
	END_REPEAT	// Init-Block. Bei Fehlern wird der Block mit EXIT vorzeitig verlassen

	// Wenn SINGLEmnParam definiert ist, dann wartet die Ausführung hier solange, bis _lSingleStep > _pl_InitState gesetzt wurde
	#ifdef SINGLEmnParam
	REPEAT
		UNTIL
		_lSingleStep > _pl_InitState OR NOT _xSingleStep
	END_REPEAT
	#endif

	// Wenn alles fehlerfrei durchgelaufen ist, wird das OK gesetzt
	// Andernfalls Meldung und Log-Datei auswerten

	IF _xSysError THEN

		_PmIntern.Status.wMsgClass := 0;
		_PmIntern.Status.wMsgNumber := MNPARAM_MSG_SYSTEMERROR;
		_PmIntern.Status.wMsgAckLevel := 255;
		_PmIntern.Status.diMsgAttr1 := 0;
		_PmIntern.Status.sMsgAttrTxt := '';

	ELSE

		//		// Aus Kompatibilitätsgründen
		//		IF PV_xgetadr(ADR('MachineState.xCfgOk'), ADR(_lAdrCfgOk), ADR(_lLenCfgOk)) = ERR_OK THEN
//
//			_xCfgOk ACCESS _lAdrCfgOk;
//			_xCfgOk := TRUE;
//
//		END_IF

		//****************************************************************************************************************
		// Ringbuffer for Logs
		//****************************************************************************************************************

		_kgRBcreatePMlog(sName := '_pmLogrb', bMemType := doTEMP, wCntEntry := 100, lLenEntry := SIZEOF(_LogEntry), wPtrWrite := _wPtrRBwrite, wPtrRead := _wPtrRBread, wPtrStart := _wPtrRBstart);

		IF _kgRBcreatePMlog.wStatus = ERR_OK THEN

			_wPtrRBloc := 0;

			_xRBReady := TRUE;

			_InsertRB.doIdent := _kgRBcreatePMlog.doIdent;
			_InsertRB.doLen := _kgRBcreatePMlog.doLen;
			_InsertRB.lLenEntry := SIZEOF(_LogEntry);
			_InsertRB.pEntry := ADR(_LogEntryIn);

			_ReadRB.doIdent := _kgRBcreatePMlog.doIdent;
			_ReadRB.doLen := _kgRBcreatePMlog.doLen;
			_ReadRB.lLenEntry := SIZEOF(_LogEntry);
			_ReadRB.pEntry := ADR(_LogEntry);

		ELSE

			_PmIntern.Logger.logLevel := arlogLEVEL_INFO;
			_PmIntern.Logger.text := 'Create Ringbuffer: {##AttrVar1}';
			_PmIntern.Logger.var1 := _kgRBcreatePMlog.wStatus;
			_PmIntern.Logger.var2 := 0;
			_PmIntern.Logger();

		END_IF

	END_IF

END_PROGRAM
```

#### mnParamExit.st
```iecst
(********************************************************************
 * COPYRIGHT -- Herbert Kannegiesser GmbH
 ********************************************************************
 * Program: mnParam
 * File: mnParamExit.st
 * Author: hunholz
 * Created: December 20, 2011
 *******************************************************************)

PROGRAM _EXIT

	IF _MemPartCreate.ident > 0 THEN

		_MemPartDestroy(enable := TRUE, ident := _MemPartCreate.ident);

	END_IF

END_PROGRAM
```

#### _mnParam.typ - Local data types
```iecst
(********************************************************************
 * COPYRIGHT -- Microsoft
 ********************************************************************
 * Program: mnParam
 * File: _mnParam.typ
 * Author: hunholz
 * Created: July 23, 2011
 ********************************************************************
 * Local data types of program mnParam
 ********************************************************************)

TYPE
	enum_CycMainState :
		(
		cs_MainIdle,
		cs_MainImport,
		cs_MainDelete,
		cs_MainWarning,
		cs_MainWaitCmdZero
		);
	enum_CycIfState :
		(
		cs_IfIdle,
		cs_IfFillEditor,
		cs_IfSaveEditor,
		cs_IfCreateIndCont,
		cs_IfDeleteIndCont,
		cs_IfCopyIndCont,
		cs_IfRestore,
		cs_IfBackup,
		cs_IfReady,
		cs_IfFillNameList
		);
	enum_CycFillEditor :
		(
		cs_feIdle,
		cs_feStart,
		cs_feFillEditor,
		cs_feRdySuccess,
		cs_feRdyFault
		);
	enum_CycSaveEditor :
		(
		cs_seIdle,
		cs_seStart,
		cs_seReadContainer,
		cs_seCommit,
		cs_seWriteDoNum,
		cs_seWriteDoString,
		cs_seWriteDoBin,
		cs_seFreeMem,
		cs_seExpCSV,
		cs_seTOC,
		cs_seRdySuccess,
		cs_seRdyFault
		);
	enum_CycImpState :
		(
		cs_ImpIdle,
		cs_ImpUSBLinkDevice,
		cs_ImpUSBStart,
		cs_ImpStart,
		cs_ImpDirInfo,
		cs_ImpShowFailed,
		cs_ImpDirRead,
		cs_ImpCheckFile,
		cs_ImpAllocMemFile,
		cs_ImpOpenFile,
		cs_ImpReadFile,
		cs_ImpCloseFile,
		cs_ImpParsVers,
		cs_ImpGetRoot,
		cs_ImpDiNum,
		cs_ImpDiNumDef,
		cs_ImpCpNum,
		cs_ImpDiStr,
		cs_ImpDiStrDef,
		cs_ImpCpStr,
		cs_ImpDiBin,
		cs_ImpDiBinDef,
		cs_ImpCpBin,
		cs_ImpAllocMemNum,
		cs_ImpAllocMemStr,
		cs_ImpRdNum,
		cs_ImpRdStr,
		cs_ImpRdBin,
		cs_ImpSetDefaultNum,
		cs_ImpSetDefaultStr,
		cs_ImpParse,
		cs_ImpFreeMemFile,
		cs_ImpWrNum,
		cs_ImpWrStr,
		cs_ImpSetPV,
		cs_ImpWrBin,
		cs_ImpFreeMemStr,
		cs_ImpFreeMemNum,
		cs_ImpExpCSV,
		cs_ImpDelDir,
		cs_ImpUSBunlinkDevice,
		cs_ImpTOC,
		cs_ImpCPCache1,
		cs_ImpCPCache2,
		cs_ImpRdyFault,
		cs_ImpRdySuccess
		);
	enum_CycDelState :
		(
		cs_DelIdle,
		cs_DelStart,
		cs_DelDInumPar,
		cs_DelDIstringPar,
		cs_DelDIbinaerPar,
		cs_DelDDnumPar,
		cs_DelDDstringPar,
		cs_DelDDbinaerPar,
		cs_DelDelFile,
		cs_DelExpToc,
		cs_DelRdyFault,
		cs_DelRdySuccess
		);
	enum_CycBackState :
		(
		cs_BacIdle,
		cs_BacUSBlinkDevice,
		cs_BacCreateDirMachine,
		cs_BacCreateDirBackup,
		cs_BacCreateDirDate,
		cs_BacCopy,
		cs_BacUSBunlinkDevice,
		cs_BacRdyFault,
		cs_BacRdySuccess
		);
	enum_CycCreateState :
		(
		cs_CrtIdle,
		cs_CrtStart,
		cs_CrtCpyNumDef,
		cs_CrtCpyStringDef,
		cs_CrtCpyBinDef,
		cs_CrtExpCSV,
		cs_CrtTOC,
		cs_CrtRdyFault,
		cs_CrtRdySuccess
		);
	enum_CycCopyState :
		(
		cs_CpyIdle,
		cs_CpyStart,
		cs_CpyChckTarget,
		cs_CpyCpyNum,
		cs_CpyCpyString,
		cs_CpyCpyBin,
		cs_CpyExpCSV,
		cs_CpyTOC,
		cs_CpyRdyFault,
		cs_CpyRdySuccess
		);
	enum_CycWriteMno :
		(
		cs_WrMnoIdle,
		cs_WrMnoDelFile,
		cs_WrMnoCreateFile,
		cs_WrMnoWriteFile,
		cs_WrMnoCloseFile,
		cs_WrMnoReset
		);
	enum_InitState :
		(
		is_DeleteImport := 10,
		is_CreateLog := 15,
		is_CreateMem := 20,
		is_TestDataModel := 40,
		is_CopyDataModel := 50,
		is_InfoDataModelDO := 60,
		is_ReadDataModel := 70,
		is_ParseDataModelVers := 80,
		is_TestVersDataModel := 90,
		is_ResetDataModel := 100,
		is_CreateTempDataModel := 110,
		is_ParseDataModel := 120,
		is_WriteDataModel := 130,
		is_TestDefautDO := 140,
		is_ResetDefaultDO := 150,
		is_CreateDefaultDO1 := 160,
		is_CreateDefaultDO2 := 161,
		is_CreateDefaultDO3 := 162,
		is_CreateDefaultDO4 := 163,
		is_CreateContainerNames := 200,
		is_LookForDOvalue := 210,
		is_LookForFile := 220,
		is_CreateDOvalue := 230,
		is_TestFileDate := 240,
		is_ImportData1 := 250,
		is_ImportData2 := 251,
		is_ImportData3 := 252,
		is_ImportData4 := 253,
		is_SetValue1 := 260,
		is_SetValue2 := 261,
		is_SetValue3 := 262,
		is_ExpCSV := 270
		);
	enum_ContainerExportState :
		(
		ces_AllocMemCSV,
		ces_CreateCSV,
		ces_DeleteFileCSV,
		ces_CreateFileCSV,
		ces_OpenFileCSV,
		ces_WriteFileCSV,
		ces_CloseFileCSV,
		ces_FreeMemCSV,
		ces_Log
		);
	enum_TocExportState :
		(
		tes_AllocMemCSV,
		tes_CreateCSV,
		tes_DeleteFileCSV,
		tes_CreateFileCSV,
		tes_OpenFileCSV,
		tes_WriteFileCSV,
		tes_CloseFileCSV,
		tes_FreeMemCSV,
		tes_Log
		);
	PmIntern_typ : 	STRUCT
		Status : kgMsg_Status_Typ;
		Logger : kgArLogWrite;
		MemSettings : MemSettings_typ;
		ExpSettings : ExpSettings_typ;
		DataModelCsv : DataModelCsv_typ;
		DataObjects : DataObjects_typ;
		CSVFile : DataModelCsv_typ;
		CSVDataObjects : CsvDataObjects_typ;
		Parse : Parse_typ;
		WriteCSV : WriteCSV_typ;
		ActContainer : Container_typ;
		ImportParamCont : DirRead_typ;
		TOC : Toc_typ;
		enInitState : enum_InitState;
		enCycMainState : enum_CycMainState;
		enCycIfState : enum_CycIfState;
		enCycImpState : enum_CycImpState;
		enCycDelState : enum_CycDelState;
		enCycFillEditor : enum_CycFillEditor;
		enCycSaveEditor : enum_CycSaveEditor;
		enCycBackup : enum_CycBackState;
		enCycCreate : enum_CycCreateState;
		enCycCopy : enum_CycCopyState;
		sActPath : STRING[63];
		sActPathAndFilename : STRING[63];
		xResetModelDOs : BOOL;
		xResetConateinerDOs : BOOL;
		xExportContainerCsv : BOOL;
	END_STRUCT;
	DirRead_typ : 	STRUCT
		lFileNumber : UDINT;
		lFileCnt : UDINT;
		fiDir_Read_Data : ARRAY[1..MNPARAM_CNT_CSVFILES]OF fiDIR_READ_DATA;
		sPcNumber : STRING[7];
	END_STRUCT;
	Container_typ : 	STRUCT
		sDoNameNum : STRING[11]; (*von Parameter Daten-Objekt*)
		sDoNameString : STRING[11]; (*von Parameter Daten-Objekt*)
		sDoNameDefNum : STRING[11];
		sDoNameDefString : STRING[11];
		sCsvName : STRING[23];
		sDoName : STRING[11]; (*von Struktur Daten-Objekt*)
		sDoNameDef : STRING[11];
		sIndex : STRING[7]; (*Index für die Instanzierung von Container Daten-Objekten*)
		sStrucRoot : STRING[31];
		lAdressStructRoot : UDINT;
		lSizeStructRoot : UDINT;
		lCountParamNum : UDINT; (*Anzahl der numerischen Parametern*)
		lCountParamString : UDINT; (*Anzahl der String-Parameter*)
		siContainerID : SINT;
		bDirect : USINT; (*0 - Indirekt*)
		wMinBound : UINT; (*Untere Grenze, bei mehreren Instanzen*)
		wDimension : UINT; (*Dimension, bei mehreren Instanzen*)
		wIndexIndirect : UINT; (*Laufindex, wenn mehrere Instanzen bearbeitet werden*)
		xDataImported : BOOL;
		xWriteProtected : BOOL;
		xExportfileExist : BOOL;
	END_STRUCT;
	ExpSettings_typ : 	STRUCT
		sCfDeviceName : STRING[10]; (*Device (Compactflash, USB-Stick)*)
		sPath : STRING[31]; (*Pfad mit abschließendem Backslash*)
		sFilename : STRING[31]; (*Dateiname*)
		sSoftwareComment : STRING[47]; (*Kommentarzeile mit Paketnamen und Version*)
		HeaderMachineNo : mnParam_HeaderMachineNoRow_typ; (*Maschinennummer*)
	END_STRUCT;
	MemSettings_typ : 	STRUCT
		PartIdent : UDINT; (*Ident der Partition*)
		PartLen : UDINT; (*Größe der Speicherpartition*)
	END_STRUCT;
	Toc_typ : 	STRUCT
		wStartIdx : ARRAY[0..MNPARAM_MAXIDX_CONTAINER]OF UINT;
		TocEntry : ARRAY[1..MNPARAM_CNT_CSVFILES]OF mnParam_CsvContent_typ;
	END_STRUCT;
	DataModelCsv_typ : 	STRUCT
		sName : STRING[23] := 'DataModel.csv'; (*Name der DatenModell.csv*)
		sNameInPm : STRING[63] := 'PM\DataModel.csv'; (*Name der DatenModell.csv im PM Ordner*)
		sNameInExp : STRING[63] := 'PM\Export\DataModel.csv'; (*Name der DatenModell.csv im Eport Ordner*)
		lAdress : UDINT;
		lSize : UDINT;
		HeaderVersion : mnParam_HeaderVersionRow_typ;
	END_STRUCT;
	DataObjects_typ : 	STRUCT
		Names : DoNames_typ;
		Idents : DoIdents_typ;
		Adress : DoIdents_typ;
		Size : DoIdents_typ;
		TempAdresses : DoIdents_typ;
		MaxIndex : DoIdents_typ;
	END_STRUCT;
	CsvDataObjects_typ : 	STRUCT
		Idents : CSVDoIdents_typ;
		Size : CSVDoIdents_typ;
		Adress : CSVDoIdents_typ;
		TempAdresses : CSVDoIdents_typ;
		MaxIndex : CSVDoIdents_typ;
	END_STRUCT;
	DoNames_typ : 	STRUCT
		sDataModelContainer : STRING[10] := '_PmCont'; (*Data Model - Container*)
		sDataModelLogicalStruct : STRING[10] := '_PmLogStru'; (*Data Model - Logische Struktur*)
		sDataModelParamNum : STRING[10] := '_PmParNum'; (*Data Model - Parameter*)
		sDataModelParamString : STRING[10] := '_PmParStr'; (*Data Model - Parameter*)
	END_STRUCT;
	DoIdents_typ : 	STRUCT
		lContainer : UDINT; (*Ident des DataObject Container*)
		lLogicalStruct : UDINT; (*Ident des DataObject Logical Struct*)
		lParamNum : UDINT; (*Ident des DataObject Param Num*)
		lParamString : UDINT; (*Ident des DataObject Param String*)
	END_STRUCT;
	CSVDoIdents_typ : 	STRUCT
		lCSVNum : UDINT;
		lCSVString : UDINT;
		lDataObjekt : UDINT;
	END_STRUCT;
	Parse_typ : 	STRUCT
		lFileAdress : UDINT;
		lFileSize : UDINT;
		lCntLines : UDINT;
		lLineTableAdress : UDINT;
		lLineTableLen : UDINT;
	END_STRUCT;
	WriteCSV_typ : 	STRUCT
		lFileSize : UDINT;
		lFileAdress : UDINT;
	END_STRUCT;
END_TYPE
```

#### _mnParam.var - Local variables
```iecst
(********************************************************************
 * COPYRIGHT -- Microsoft
 ********************************************************************
 * Program: mnParam
 * File: _mnParam.var
 * Author: hunholz
 * Created: July 23, 2011
 ********************************************************************
 * Local variables of program mnParam
 ********************************************************************)
(*Konstanten*)
(*Single Step*)
VAR
	_xSingleStep : BOOL;
	_lSingleStep : UDINT := 0;
	_wSinglestep : UINT := 0;
END_VAR
(*Debug*)
VAR
	_xDebug : BOOL;
	_xWeiter : BOOL;
	_pl_InitState : REFERENCE TO UDINT;
END_VAR
(*Ergebnisse des InitUp*)
VAR
	_xInitOk : BOOL; (*Bleibt solange TRUE, wie es keinen Fehler in der Initialisierung gegeben hat*)
END_VAR
(*Statusvariablen*)
VAR
	_xAllContainerOK : BOOL;
END_VAR
(*Temporärer Speicher*)
VAR
	_MemPartCreate : AsMemPartCreate;
	_MemPartAlloc : AsMemPartAllocClear;
	_MemPartFree : AsMemPartFree;
END_VAR
(*Von Markus verwendete Variablen*)
VAR
	_PmIntern : PmIntern_typ;
END_VAR
(*Parsetable*)
VAR
	_plLineAdress : REFERENCE TO ARRAY[1..MNPARAM_MAXPARSELINES] OF UDINT;
	_pwLineLen : REFERENCE TO ARRAY[1..MNPARAM_MAXPARSELINES] OF UINT;
	_CountLines : mnParam_CountLines;
	_wStartLine : UINT;
	_GetCsvDat : mnParam_GetCsvDat;
END_VAR
(*Allgemeine Fileoperationen*)
VAR
	_FileOpen : FileOpen;
	_FileInfo : FileInfo;
	_fiFileInfo : fiFILE_INFO;
	_FileCopy : FileCopy;
	_FileRead : FileRead;
	_FileClose : FileClose;
END_VAR
(*Datenmodell Datenobjekte*)
VAR
	_diContainer : DatObjInfo;
	_diLogicalStruct : DatObjInfo;
	_diParamNum : DatObjInfo;
	_diParamString : DatObjInfo;
	_ddContainer : DatObjDelete;
	_ddLogicalStruct : DatObjDelete;
	_ddParamNum : DatObjDelete;
	_ddParamString : DatObjDelete;
	_dcContainer : DatObjCreate;
	_dcLogicalStruct : DatObjCreate;
	_dcParamString : DatObjCreate;
	_dcParamNum : DatObjCreate;
	_pDoContainer : REFERENCE TO mnParam_ContainerDyn_typ;
	_pDoLogicalStruct : REFERENCE TO mnParam_LogicalStructDyn_typ;
	_pDoParamNum : REFERENCE TO mnParam_ParamNumDyn_typ;
	_pDoParamString : REFERENCE TO mnParam_ParamStringDyn_typ;
	_wIndex : UINT;
END_VAR
(*CSV Datenobjekte*)
VAR
	_diCSVNum : DatObjInfo;
	_diCSVString : DatObjInfo;
	_diDefaultDO : DatObjInfo;
	_diDO : DatObjInfo;
	_drDO : DatObjRead;
	_ddCSVNum : DatObjDelete;
	_ddCSVString : DatObjDelete;
	_ddDataObjekt : DatObjDelete;
	_dcCSVNum : DatObjCreate;
	_dcCSVString : DatObjCreate;
	_dcDataObjekt : DatObjCreate;
	_pDoContainerNum : REFERENCE TO mnParam_CsvNumDyn_typ;
	_pDoContainerString : REFERENCE TO mnParam_CsvStringDyn_typ;
END_VAR
(*Datencontainer*)
VAR
	_c : DINT;
	_sIndex : STRING[3];
END_VAR
(*Struct-Root Erkennung*)
VAR
	_lPVadress : UDINT;
	_lPVlen : UDINT;
END_VAR
(*CSV-Daten erzeugen*)
VAR
	_getContainerParamNum : mnParam_GetContainerOfParamNum;
	_getContainerParamString : mnParam_GetContainerOfParamStrin;
	_wIdxCsvNum : UINT;
	_wIdxCsvString : UINT;
	_i1 : UINT;
	_i2 : UINT;
	_i3 : UINT;
	_i4 : UINT;
	_dim1 : UINT;
	_dim2 : UINT;
	_dim3 : UINT;
	_dim4 : UINT;
	_i : UINT;
	_sPVAdress : STRING[63];
	_WritePVNum : mnParam_WritePVNum;
	_WritePVString : mnParam_WritePVString;
	_wDimension : UINT;
	_dcpCSVNum : DatObjCopy;
	_dcpCSVString : DatObjCopy;
	_dcpDefaultDO : DatObjCopy;
	_xFoundVersion : BOOL;
	_xFoundDate : BOOL;
	_CsvHeaderVersion : mnParam_HeaderVersionRow_typ;
	_CsvHeaderDate : mnParam_HeaderTimeRow_typ;
	_drCSVNum : DatObjRead;
	_drCSVString : DatObjRead;
	_binarySearchNum : mnParam_BinarySearchInNumeric;
	_binarySearchString : mnParam_BinarySearchInString;
	_dwCSVNum : DatObjWrite;
	_DTGetTime : DTGetTime;
	_dwCSVString : DatObjWrite;
	_wStatus : UINT;
	_PN : mnParam_ParamNumRow_typ;
	_CN : mnParam_CsvNumRow_typ;
	_PS : mnParam_ParamStringRow_typ;
	_CS : mnParam_CsvStringRow_typ;
	_dwDO : DatObjWrite;
	_sNumeric : STRING[11];
	TONwarn : TON;
	_FileDelete : FileDelete;
	_DirRead : DirRead;
	_xFoundFile : BOOL;
	_xFoundMachineNo : BOOL;
	_CsvHeadMachineNo : mnParam_HeaderMachineNoRow_typ;
	_dtStartSetPV : DATE_AND_TIME;
	_dtEndSetPV : DATE_AND_TIME;
	_WritePVrNum : mnParam_WritePVrNum;
	_pdiValue : REFERENCE TO DINT;
	_rValue : REAL;
	_DirDeleteEx : DirDeleteEx;
	_sPathMnrCsv : STRING[31];
	_FileOpenCsv : FileOpen;
	_utfParseMem : ARRAY[0..127] OF UINT;
	_FileReadCsv : FileRead;
	_lPosLF : UDINT;
	_lPosCR : UDINT;
	_FileCloseCsv : FileClose;
	_AsArLogCreate : AsArLogCreate;
	_AsArLogGetInfo : AsArLogGetInfo;
	_xSysError : BOOL := FALSE;
	_DirCreate : DirCreate;
	_MemPartDestroy : AsMemPartDestroy;
	_lAdrInfoMaschinennummer : UDINT;
	_lLenInfoMaschinennummer : UDINT;
	_utfMaschinennummer : REFERENCE TO WSTRING[15];
	_lAdrInfoMaschinentyp : UDINT;
	_lLenInfoMaschinentyp : UDINT;
	_utfMaschinentyp : REFERENCE TO WSTRING[15];
	_sPkgName : STRING[11];
	_VerStruc : MoVerStruc_typ;
	_lLineMem : UDINT;
	_lModelMem : UDINT;
	_lContMem : UDINT;
	_ec : _ExportContainer;
	_wIdxToc : UINT;
	_ExportTableOfContent : _ExportToc;
	_DefineActContainer : _DefActContainer;
	_wIndexIndirect : UINT;
	_EditNumValues : mnParam_EditNumValue_typ;
	_EditStrValues : mnParam_EditStrValue_typ;
	_wActRow : UINT;
	_wActIdx : UINT;
	_GetAccessRights : _GetRights;
	_wActRefIdx : UINT;
	_prValue : REFERENCE TO REAL;
	_pFunctionTxt : REFERENCE TO ARRAY[0..MNTXT_MAX_IDX_TXT_FUNCTION] OF mnTxt_TxtLine_Typ;
	_pInstanceTxt : REFERENCE TO ARRAY[0..MNTXT_MAX_IDX_TXT_INSTANCE] OF mnTxt_TxtLine_Typ;
	_pParamTxt : REFERENCE TO ARRAY[0..MNTXT_MAX_IDX_TXT_PARAMETER] OF mnTxt_TxtLine_Typ;
	_pParamHlpTxt : REFERENCE TO ARRAY[0..MNTXT_MAX_IDX_TXT_PARAMETER] OF mnTxt_HelpTxtLine_Typ;
	_wIdxFunctionTxt : UINT;
	_wIdxInstanceTxt : UINT;
	_wIdxParamTxt : UINT;
	_wIdxParamHlpTxt : UINT;
	_wLenUtf : UINT;
	_pDigits : UDINT;
	_xNumDirty : BOOL;
	_xStrDirty : BOOL;
	_pUnit : UDINT;
	_ii : USINT;
	_prMinValue : REFERENCE TO REAL;
	_prMaxValue : REFERENCE TO REAL;
	_wDelCont : UINT;
	_wDelInst : UINT;
	_xImpSetDefault : BOOL;
	_DirInfo : DirInfo;
	_xFoundOneFile : BOOL;
	_LogEntry : KG_ErrLog_typ;
	_wPtrRBwrite : UINT;
	_wPtrRBread : UINT;
	_wPtrRBstart : UINT;
	_kgRBcreatePMlog : kgRBcreate;
	_wPtrRBloc : UINT;
	_xRBReady : BOOL;
	_InsertRB : kgRBinsert;
	_LogEntryIn : KG_ErrLog_typ;
	_ReadRB : kgRBread;
	_wLogStep : UINT;
	_xNextFile : BOOL;
END_VAR
VAR CONSTANT
	_MNPARAM_LOG_STARTIMPORT : UINT := 1;
	_MNPARAM_LOG_STARTDELETE : UINT := 2;
	_MNPARAM_LOG_ENDIMPORT_SUCC : UINT := 3;
	_MNPARAM_LOG_ENDIMPORT_FAILED : UINT := 4;
	_MNPARAM_LOG_ENDDELETE_SUCC : UINT := 5;
	_MNPARAM_LOG_ENDDELETE_FAILED : UINT := 6;
	_MNPARAM_LOG_STARTSAVE : UINT := 7;
	_MNPARAM_LOG_ENDSAVE_SUCC : UINT := 8;
	_MNPARAM_LOG_ENDSAVE_FAILED : UINT := 9;
	_MNPARAM_LOG_FOUNDFILES : UINT := 10;
	_MNPARAM_LOG_FOUNDFILE : UINT := 11;
	_MNPARAM_LOG_WRONGMACHINENO : UINT := 12;
	_MNPARAM_LOG_WRONGMACHINETYPE : UINT := 13;
	_MNPARAM_LOG_NOVERSION : UINT := 14;
	_MNPARAM_LOG_CNTLINES : UINT := 15;
	_MNPARAM_LOG_WRITEPROTECTED : UINT := 16;
	_MNPARAM_LOG_SYSTEMFAULT : UINT := 17;
	_MNPARAM_LOG_STARTRESTORE : UINT := 18;
	_MNPARAM_LOG_STARTBACKUP : UINT := 19;
	_MNPARAM_LOG_ENDRESTORE_SUCC : UINT := 20;
	_MNPARAM_LOG_ENDRESTORE_FAILED : UINT := 21;
	_MNPARAM_LOG_ENDBACKUP_SUCC : UINT := 22;
	_MNPARAM_LOG_ENDBACKUP_FAILED : UINT := 23;
	_MNPARAM_LOG_STARTCREATE : UINT := 24;
	_MNPARAM_LOG_ENDCREATE_SUCC : UINT := 25;
	_MNPARAM_LOG_ENDCREATE_FAILED : UINT := 26;
	_MNPARAM_LOG_STARTCOPY : UINT := 27;
	_MNPARAM_LOG_ENDCOPY_SUCC : UINT := 28;
	_MNPARAM_LOG_ENDCOPY_FAILED : UINT := 29;
	_MNPARAM_LOG_ROOTVAR : UINT := 30;
	_MNPARAM_LOG_FOUNDIMPDIR : UINT := 31;
END_VAR
VAR
	_CsvHeaderMachineNo : mnParam_HeaderMachineNoRow_typ;
	_sUSBInterface : STRING[31];
END_VAR
VAR CONSTANT
	_MNPARAM_TEMP_USBDEV : STRING[15] := 'TEMPUSB';
END_VAR
VAR
	_DevLink : DevLink;
	_sDevString : STRING[63];
	_DevUnlink : DevUnlink;
	_sImportDevice : STRING[31];
	_lDevLinkHandle : UDINT;
	_GetBackupTime : DTGetTime;
	_BackupTimestamp : mnParam_datetoa;
	_DirCopy : DirCopy;
	_wCreateCont : UINT;
	_wCreateInst : UINT;
	_wCopyCont : UINT;
	_wCopyInst : UINT;
	_wCopyInstFrom : UINT;
	_xAllowCommands : BOOL;
	_wImpSource : UINT;
	TONwarn2 : TON;
	_wActListIdx : UINT;
	_k : UINT;
	_diProgname : DatObjInfo;
	_pDoProgContainer : REFERENCE TO mnParam_CsvStringDyn_typ;
	_lMaxIndexProgContainer : UDINT;
	_TONshowfailed : TON;
	_inst : UINT;
	_xParamOK : BOOL;
	_wStateImportDatamodel : UINT;
	_xFoundDM : BOOL;
	_lDirNum : UDINT;
	_sTestFile : STRING[63];
	_xImpDMOK : BOOL;
	_xModelImportChecked : BOOL;
	_fiDataModel : fiFILE_INFO;
	_fiMNR : fiFILE_INFO;
	_LP : _LimParam;
	_wCntParams : UINT;
	_xRun : BOOL;
	_lLoop : UDINT;
	_lLoopCount : UDINT;
	_xNoWriteProtect : BOOL;
	_cycStateWriteMno : enum_CycWriteMno;
	_FileMnoDelete : FileDelete;
	_FileMnoCreate : FileCreate;
	_bBufMno : ARRAY[0..47] OF USINT;
	_lAdrBuf : UDINT;
	_lSizeBuf : UDINT;
	_WriteBOM : mnParam_WriteBOM_Mem;
	_WriteMno : mnParam_WriteCSV252_Mem;
	_newMno : mnParam_HeaderMachineNoRow_typ;
	_FileMnoWrite : FileWrite;
	_FileMnoClose : FileClose;
END_VAR
```

#### _ExportContainer.st - Schreibe Containerdaten in eine CSV-Datei
```iecst
(********************************************************************
 * COPYRIGHT -- Herbert Kannegiesser GmbH
 ********************************************************************
 * Program: mnParam
 * File: _ExportContainer.st
 * Author: hunholz
 * Created: February 16, 2012
 ********************************************************************
 * Implementation of program mnParam
 ********************************************************************)

(* Schreibe Containerdaten in eine CSV-Datei *)
FUNCTION_BLOCK _ExportContainer

	IF Enable THEN

		Status := ERR_OK;

		//=======================
		// Auf Nullpointer prüfen
		//=======================

		IF pIntern = 0 THEN
			Status := MNPARAM_STAT_NULLPOINTER;
			RETURN;
		END_IF

		_Intern ACCESS pIntern;

		IF _Intern.DataObjects.Adress.lContainer = 0 THEN
			Status := MNPARAM_STAT_NULLPOINTER;
			RETURN;
		END_IF

		_DoContainer ACCESS _Intern.DataObjects.Adress.lContainer;

		IF _Intern.DataObjects.Adress.lParamNum = 0 THEN
			Status := MNPARAM_STAT_NULLPOINTER;
			RETURN;
		END_IF

		_DoParamNum ACCESS _Intern.DataObjects.Adress.lParamNum;

		IF _Intern.DataObjects.Adress.lParamString = 0 THEN
			Status := MNPARAM_STAT_NULLPOINTER;
			RETURN;
		END_IF

		_DoParamString ACCESS _Intern.DataObjects.Adress.lParamString;

		IF _Intern.CSVDataObjects.Adress.lCSVNum = 0 THEN
			Status := MNPARAM_STAT_NULLPOINTER;
			RETURN;
		END_IF

		_DoNum ACCESS _Intern.CSVDataObjects.Adress.lCSVNum;

		IF _Intern.CSVDataObjects.Adress.lCSVString = 0 THEN
			Status := MNPARAM_STAT_NULLPOINTER;
			RETURN;
		END_IF

		_DoString ACCESS _Intern.CSVDataObjects.Adress.lCSVString;

		//===================
		// Eigentliche Aktion
		//===================

		_xReady := FALSE;
		_xBusy := FALSE;

		REPEAT

			CASE _ContainerExpState OF

				//=============================================
				// Speicher zum schreiben der Zeilen allokieren
				//=============================================
				ces_AllocMemCSV:

					_wIntStatus := 0;

					_MemPartAlloc(enable := TRUE, ident := _Intern.MemSettings.PartIdent , len := MNPARAM_TEMPWRITECSVSIZE);

					IF _MemPartAlloc.status = ERR_OK THEN

						_Intern.WriteCSV.lFileAdress := _MemPartAlloc.mem;
						_Intern.WriteCSV.lFileSize := 0;

						_ContainerExpState := ces_CreateCSV;

						_xFault := FALSE;

					ELSIF _MemPartAlloc.status <> ERR_FUB_BUSY THEN

						_wIntStatus := MNPARAM_STAT_EXPALLOCMEMCSV;
						_wIntAdStatus := _MemPartAlloc.status;

						_ContainerExpState := ces_Log;

						_Intern.Logger.logLevel := arlogLEVEL_INFO;
						_Intern.Logger.text		:= 'MemPartAlloc for Writing CSV File for Container Index: {##AttrVar1}. Status : {##AttrVar2}';
						_Intern.Logger.var1		:= _Intern.ActContainer.siContainerID;
						_Intern.Logger.var2		:= _MemPartAlloc.status;

					ELSE

						_xBusy := TRUE;

					END_IF

				//=============================================
				// Zeilen schreiben
				//=============================================
				ces_CreateCSV:

					_WriteBOM(enable := TRUE, pMem := _Intern.WriteCSV.lFileAdress, lMaxSize := MNPARAM_TEMPWRITECSVSIZE, lSize := _Intern.WriteCSV.lFileSize);

					// Kopfdaten schreiben
					_WriteComment(enable := TRUE, pMem := _Intern.WriteCSV.lFileAdress, lMaxSize := MNPARAM_TEMPWRITECSVSIZE, sComment := _Intern.ExpSettings.sSoftwareComment , lSize := _Intern.WriteCSV.lFileSize);
					_WriteNewLine(enable := TRUE, pMem := _Intern.WriteCSV.lFileAdress, lMaxSize := MNPARAM_TEMPWRITECSVSIZE, lSize := _Intern.WriteCSV.lFileSize);

					_WriteVersion(enable := TRUE, pMem := _Intern.WriteCSV.lFileAdress, lMaxSize := MNPARAM_TEMPWRITECSVSIZE, VersionRow := _Intern.DataModelCsv.HeaderVersion, lSize := _Intern.WriteCSV.lFileSize);

					_WriteNewLine(enable := TRUE, pMem := _Intern.WriteCSV.lFileAdress, lMaxSize := MNPARAM_TEMPWRITECSVSIZE, lSize := _Intern.WriteCSV.lFileSize);

					_WriteMachineNo(enable := TRUE, pMem := _Intern.WriteCSV.lFileAdress, lMaxSize := MNPARAM_TEMPWRITECSVSIZE, MachineNoRow := _Intern.ExpSettings.HeaderMachineNo, lSize := _Intern.WriteCSV.lFileSize);

					_WriteNewLine(enable := TRUE, pMem := _Intern.WriteCSV.lFileAdress, lMaxSize := MNPARAM_TEMPWRITECSVSIZE, lSize := _Intern.WriteCSV.lFileSize);

					_WriteTimeStamp(enable := TRUE, pMem := _Intern.WriteCSV.lFileAdress, lMaxSize := MNPARAM_TEMPWRITECSVSIZE, TimeRow := _DoNum.Header.Time, lSize := _Intern.WriteCSV.lFileSize);

					_WriteNewLine(enable := TRUE, pMem := _Intern.WriteCSV.lFileAdress, lMaxSize := MNPARAM_TEMPWRITECSVSIZE, lSize := _Intern.WriteCSV.lFileSize);

					_WriteComment(enable := TRUE, pMem := _Intern.WriteCSV.lFileAdress, lMaxSize := MNPARAM_TEMPWRITECSVSIZE, sComment := 'Numeric Parameter:', lSize := _Intern.WriteCSV.lFileSize);

					_WriteNewLine(enable := TRUE, pMem := _Intern.WriteCSV.lFileAdress, lMaxSize := MNPARAM_TEMPWRITECSVSIZE, lSize := _Intern.WriteCSV.lFileSize);

					// Numerische Daten schreiben

					_wOldIdx := 65535;

					FOR _i := 1 TO UDINT_TO_UINT(_Intern.CSVDataObjects.MaxIndex.lCSVNum) DO

						IF _DoNum.CsvNum[_i].xChanged THEN

							IF _wOldIdx <> _DoNum.CsvNum[_i].wIdxNumPar THEN

								_wOldIdx := _DoNum.CsvNum[_i].wIdxNumPar;

								_WriteNewLine(enable := TRUE, pMem := _Intern.WriteCSV.lFileAdress, lMaxSize := MNPARAM_TEMPWRITECSVSIZE, lSize := _Intern.WriteCSV.lFileSize);

								_WriteComment(enable := TRUE, pMem := _Intern.WriteCSV.lFileAdress, lMaxSize := MNPARAM_TEMPWRITECSVSIZE, sComment := _DoParamNum.ParamNum[_wOldIdx].sAdresse, lSize := _Intern.WriteCSV.lFileSize);

							END_IF

							IF _DoNum.CsvNum[_i].bRowType = 0 THEN

								_WriteNumPar(enable := TRUE, pMem := _Intern.WriteCSV.lFileAdress, lMaxSize := MNPARAM_TEMPWRITECSVSIZE, NumRow := _DoNum.CsvNum[_i], lSize := _Intern.WriteCSV.lFileSize);

							ELSE

								_WriteRealPar(enable := TRUE, pMem := _Intern.WriteCSV.lFileAdress, lMaxSize := MNPARAM_TEMPWRITECSVSIZE, NumRow := _DoNum.CsvNum[_i], lSize := _Intern.WriteCSV.lFileSize);

							END_IF

						END_IF

					END_FOR

					_WriteNewLine(enable := TRUE, pMem := _Intern.WriteCSV.lFileAdress, lMaxSize := MNPARAM_TEMPWRITECSVSIZE, lSize := _Intern.WriteCSV.lFileSize);

					_WriteComment(enable := TRUE, pMem := _Intern.WriteCSV.lFileAdress, lMaxSize := MNPARAM_TEMPWRITECSVSIZE, sComment := 'String Parameter:', lSize := _Intern.WriteCSV.lFileSize);

					_WriteNewLine(enable := TRUE, pMem := _Intern.WriteCSV.lFileAdress, lMaxSize := MNPARAM_TEMPWRITECSVSIZE, lSize := _Intern.WriteCSV.lFileSize);

					// String Daten schreiben

					_wOldIdx := 65535;

					FOR _i := 1 TO UDINT_TO_UINT(_Intern.CSVDataObjects.MaxIndex.lCSVString) DO

						IF _DoString.CsvString[_i].xChanged THEN

							IF _wOldIdx <> _DoString.CsvString[_i].wIdxStringPar THEN

								_wOldIdx := _DoString.CsvString[_i].wIdxStringPar;

								_WriteNewLine(enable := TRUE, pMem := _Intern.WriteCSV.lFileAdress, lMaxSize := MNPARAM_TEMPWRITECSVSIZE, lSize := _Intern.WriteCSV.lFileSize);

								_WriteComment(enable := TRUE, pMem := _Intern.WriteCSV.lFileAdress, lMaxSize := MNPARAM_TEMPWRITECSVSIZE, sComment := _DoParamString.ParamString[_wOldIdx].sAdresse, lSize := _Intern.WriteCSV.lFileSize);

							END_IF

							_WriteString(enable := TRUE, pMem := _Intern.WriteCSV.lFileAdress, lMaxSize := MNPARAM_TEMPWRITECSVSIZE, StringRow := _DoString.CsvString[_i], lSize := _Intern.WriteCSV.lFileSize);

						END_IF

					END_FOR

					_WriteFileEnd(enable := TRUE, pMem := _Intern.WriteCSV.lFileAdress, lMaxSize := MNPARAM_TEMPWRITECSVSIZE, lSize := _Intern.WriteCSV.lFileSize);

					_ContainerExpState := ces_DeleteFileCSV;

					_sPathAndFilename := CONCAT(_Intern.ExpSettings.sPath, _Intern.ExpSettings.sFilename);

				//==============================================
				// Möglicherweise vorhandene Exportdatei löschen
				//==============================================
				ces_DeleteFileCSV:

					_deleteCSVFile(enable := TRUE, pDevice := ADR(_Intern.ExpSettings.sCfDeviceName), pName := ADR(_sPathAndFilename));

					IF _deleteCSVFile.status <> ERR_FUB_BUSY THEN

						_ContainerExpState := ces_CreateFileCSV;

					ELSE

						_xBusy := TRUE;

					END_IF

				//==============================================
				// Exportdatei erzeugen
				//==============================================
				ces_CreateFileCSV:

					_createCSVFile(enable := TRUE, pDevice := ADR(_Intern.ExpSettings.sCfDeviceName), pFile := ADR(_sPathAndFilename) );

					IF _createCSVFile.status = ERR_OK THEN

						_ContainerExpState := ces_WriteFileCSV;
//						_ContainerExpState := ces_OpenFileCSV;

					ELSIF _createCSVFile.status <> ERR_FUB_BUSY THEN

						_wIntStatus := MNPARAM_STAT_CREATECSV;
						_wIntAdStatus := _createCSVFile.status;

						_ContainerExpState := ces_FreeMemCSV;

						_Intern.Logger.logLevel 	:= arlogLEVEL_INFO;
						_Intern.Logger.text		:= 'FileCreate for Writing CSV File for Container Index: {##AttrVar1}. Status : {##AttrVar2}';
						_Intern.Logger.var1		:= _Intern.ActContainer.siContainerID;
						_Intern.Logger.var2		:= _createCSVFile.status;

						_xFault := TRUE;

					ELSE

						_xBusy := TRUE;

					END_IF

				//==============================================
				// Exportdatei öffnen
				//==============================================
				ces_OpenFileCSV:

					_openCSVFile(enable := TRUE, pDevice := ADR(_Intern.ExpSettings.sCfDeviceName), pFile := ADR(_sPathAndFilename), mode := fiWRITE_ONLY);

					IF _openCSVFile.status = ERR_OK THEN

						_ContainerExpState := ces_WriteFileCSV;

					ELSIF _openCSVFile.status <> ERR_FUB_BUSY THEN

						_wIntStatus := MNPARAM_STAT_OPENCSV;
						_wIntAdStatus := _openCSVFile.status;

						_ContainerExpState := ces_FreeMemCSV;

						_Intern.Logger.logLevel := arlogLEVEL_INFO;
						_Intern.Logger.text		:= 'FileOpen for Writing CSV File for Container Index: {##AttrVar1}. Status : {##AttrVar2}';
						_Intern.Logger.var1		:= _Intern.ActContainer.siContainerID;
						_Intern.Logger.var2		:= _openCSVFile.status;

						_xFault := TRUE;

					ELSE

						_xBusy := TRUE;

					END_IF

				//==============================================
				// Exportdatei schreiben
				//==============================================
				ces_WriteFileCSV:

					_writeCSVFile(enable := TRUE, ident := _createCSVFile.ident, offset := 0, pSrc :=_Intern.WriteCSV.lFileAdress, len := _Intern.WriteCSV.lFileSize);

					IF _writeCSVFile.status = ERR_OK THEN

						_ContainerExpState := ces_CloseFileCSV;

						_DTGetTime(enable := TRUE);
						dtContainerWritten := _DTGetTime.DT1;

						_wIdxToc := _Intern.TOC.wStartIdx[_Intern.ActContainer.siContainerID * (-1)] + _Intern.ActContainer.wIndexIndirect - _Intern.ActContainer.wMinBound;

						IF _wIdxToc >= 1 AND _wIdxToc <= MNPARAM_CNT_CSVFILES THEN
							_Intern.TOC.TocEntry[_wIdxToc].dtTimestamp := _DoNum.Header.Time.dtTimestamp;
						END_IF

					ELSIF _writeCSVFile.status <> ERR_FUB_BUSY THEN

						_wIntStatus := MNPARAM_STAT_WRITECSV;
						_wIntAdStatus := _writeCSVFile.status;

						_ContainerExpState := ces_CloseFileCSV;

						_Intern.Logger.logLevel := arlogLEVEL_INFO;
						_Intern.Logger.text		:= 'FileWrite for Writing CSV File for Container Index: {##AttrVar1}. Status : {##AttrVar2}';
						_Intern.Logger.var1		:= _Intern.ActContainer.siContainerID;
						_Intern.Logger.var2		:= _writeCSVFile.status;

						_xFault := TRUE;

					ELSE

						_xBusy := TRUE;

					END_IF

				//==============================================
				// Exportdatei schließen
				//==============================================
				ces_CloseFileCSV:

					_closeCSVFile(enable := TRUE, ident := _createCSVFile.ident);

					IF _closeCSVFile.status = ERR_OK THEN

						_ContainerExpState := ces_FreeMemCSV;

					ELSIF _closeCSVFile.status <> ERR_FUB_BUSY THEN

						IF NOT _xFault THEN

							_wIntStatus := MNPARAM_STAT_CLOSECSV;
							_wIntAdStatus := _closeCSVFile.status;

							_Intern.Logger.logLevel := arlogLEVEL_INFO;
							_Intern.Logger.text		:= 'FileClose for Writing CSV File for Container Index: {##AttrVar1}. Status : {##AttrVar2}';
							_Intern.Logger.var1		:= _Intern.ActContainer.siContainerID;
							_Intern.Logger.var2		:= _closeCSVFile.status;

						END_IF

						_xFault := TRUE;

						_ContainerExpState := ces_FreeMemCSV;

					ELSE

						_xBusy := TRUE;

					END_IF

				//==============================================
				// Allokierten Speicher frei geben
				//==============================================
				ces_FreeMemCSV:

					_MemPartFree(enable := TRUE, ident  := _Intern.MemSettings.PartIdent, mem := _Intern.WriteCSV.lFileAdress);

					IF _MemPartFree.status = ERR_OK THEN

						_Intern.WriteCSV.lFileAdress := 0;
						_Intern.WriteCSV.lFileSize := 0;

						IF _xFault THEN

							Status := _wIntStatus;
							AdStatus := _wIntAdStatus;

							_ContainerExpState := ces_Log;

						ELSE

							Status := ERR_OK;
							AdStatus := 0;

							_xReady := TRUE;

							_ContainerExpState := ces_AllocMemCSV;

						END_IF

					ELSIF _MemPartFree.status <> ERR_FUB_BUSY THEN

						_Intern.WriteCSV.lFileAdress := 0;
						_Intern.WriteCSV.lFileSize := 0;

						IF _xFault THEN

							Status := _wIntStatus;
							AdStatus := _wIntAdStatus;

						ELSE

							Status := MNPARAM_STAT_EXPFREEMEM;
							AdStatus := _MemPartFree.status;

							_Intern.Logger.logLevel := arlogLEVEL_INFO;
							_Intern.Logger.text		:= 'FreeMem for Writing CSV File for Container Index: {##AttrVar1}. Status : {##AttrVar2}';
							_Intern.Logger.var1		:= _Intern.ActContainer.siContainerID;
							_Intern.Logger.var2		:= _MemPartFree.status;

						END_IF

						_ContainerExpState := ces_Log;

					ELSE

						_xBusy := TRUE;

					END_IF

				//==============
				// Fehler loggen
				//==============
				ces_Log:

					_Intern.Logger();

					IF _Intern.Logger.status <> ERR_FUB_BUSY THEN

						Status := _wIntStatus;
						AdStatus := _wIntAdStatus;

						_ContainerExpState := ces_AllocMemCSV;

						_xReady := TRUE;

					ELSE

						_xBusy := TRUE;

					END_IF

			END_CASE

			UNTIL

			_xBusy OR _xReady

		END_REPEAT

		IF _xBusy THEN
			Status := ERR_FUB_BUSY;
		END_IF

	ELSE

		_ContainerExpState := ces_AllocMemCSV;

		Status := ERR_FUB_ENABLE_FALSE;
		AdStatus := 0;

	END_IF

END_FUNCTION_BLOCK
```

#### _ExportToc.st - Inhaltsverzeichnis schreiben
```iecst
(********************************************************************
 * COPYRIGHT -- Herbert Kannegiesser GmbH
 ********************************************************************
 * Program: mnParam
 * File: _ExportToc.st
 * Author: hunholz
 * Created: February 16, 2012
 ********************************************************************
 * Implementation of program mnParam
 ********************************************************************)

(* Inhaltsverzeichnis schreiben *)
FUNCTION_BLOCK _ExportToc

	IF Enable THEN

		Status := ERR_OK;

		//=======================
		// Auf Nullpointer prüfen
		//=======================

		IF pIntern = 0 THEN
			Status := MNPARAM_STAT_NULLPOINTER;
			RETURN;
		END_IF

		_Intern ACCESS pIntern;

		//===================
		// Eigentliche Aktion
		//===================

		_xReady := FALSE;
		_xBusy := FALSE;

		REPEAT

			CASE _TocExpState OF

				//=============================================
				// Speicher zum schreiben der Zeilen allokieren
				//=============================================
				tes_AllocMemCSV:

					_wIntStatus := 0;

					_MemPartAlloc(enable := TRUE, ident := _Intern.MemSettings.PartIdent , len := MNPARAM_TEMPWRITECSVSIZE);

					IF _MemPartAlloc.status = ERR_OK THEN

						_Intern.WriteCSV.lFileAdress := _MemPartAlloc.mem;
						_Intern.WriteCSV.lFileSize := 0;

						_TocExpState := tes_CreateCSV;

						_xFault := FALSE;

					ELSIF _MemPartAlloc.status <> ERR_FUB_BUSY THEN

						_wIntStatus := MNPARAM_STAT_EXPALLOCMEMCSV;
						_wIntAdStatus := _MemPartAlloc.status;

						_TocExpState := tes_Log;

						_Intern.Logger.logLevel := arlogLEVEL_INFO;
						_Intern.Logger.text		:= 'MemPartAlloc for Writing TOC File : {##AttrVar2}';
						_Intern.Logger.var1		:= 0;
						_Intern.Logger.var2		:= _MemPartAlloc.status;

					ELSE

						_xBusy := TRUE;

					END_IF

				//=============================================
				// Zeilen schreiben
				//=============================================
				ces_CreateCSV:

					_WriteBOM(enable := TRUE, pMem := _Intern.WriteCSV.lFileAdress, lMaxSize := MNPARAM_TEMPWRITECSVSIZE, lSize := _Intern.WriteCSV.lFileSize);

					// Kopfdaten schreiben
					_WriteComment(enable := TRUE, pMem := _Intern.WriteCSV.lFileAdress, lMaxSize := MNPARAM_TEMPWRITECSVSIZE, sComment := _Intern.ExpSettings.sSoftwareComment , lSize := _Intern.WriteCSV.lFileSize);
					_WriteNewLine(enable := TRUE, pMem := _Intern.WriteCSV.lFileAdress, lMaxSize := MNPARAM_TEMPWRITECSVSIZE, lSize := _Intern.WriteCSV.lFileSize);

					_WriteVersion(enable := TRUE, pMem := _Intern.WriteCSV.lFileAdress, lMaxSize := MNPARAM_TEMPWRITECSVSIZE, VersionRow := _Intern.DataModelCsv.HeaderVersion, lSize := _Intern.WriteCSV.lFileSize);

					_WriteNewLine(enable := TRUE, pMem := _Intern.WriteCSV.lFileAdress, lMaxSize := MNPARAM_TEMPWRITECSVSIZE, lSize := _Intern.WriteCSV.lFileSize);

					_WriteMachineNo(enable := TRUE, pMem := _Intern.WriteCSV.lFileAdress, lMaxSize := MNPARAM_TEMPWRITECSVSIZE, MachineNoRow := _Intern.ExpSettings.HeaderMachineNo, lSize := _Intern.WriteCSV.lFileSize);

					_WriteNewLine(enable := TRUE, pMem := _Intern.WriteCSV.lFileAdress, lMaxSize := MNPARAM_TEMPWRITECSVSIZE, lSize := _Intern.WriteCSV.lFileSize);

					_DTGetTime(enable := TRUE);
					_HeaderTimeRow.dtTimestamp := _DTGetTime.DT1;
					dtTocWritten := _DTGetTime.DT1;

					_WriteTimeStamp(enable := TRUE, pMem := _Intern.WriteCSV.lFileAdress, lMaxSize := MNPARAM_TEMPWRITECSVSIZE, TimeRow := _HeaderTimeRow, lSize := _Intern.WriteCSV.lFileSize);

					_WriteNewLine(enable := TRUE, pMem := _Intern.WriteCSV.lFileAdress, lMaxSize := MNPARAM_TEMPWRITECSVSIZE, lSize := _Intern.WriteCSV.lFileSize);

					_WriteComment(enable := TRUE, pMem := _Intern.WriteCSV.lFileAdress, lMaxSize := MNPARAM_TEMPWRITECSVSIZE, sComment := 'Table Of Content', lSize := _Intern.WriteCSV.lFileSize);

					_WriteNewLine(enable := TRUE, pMem := _Intern.WriteCSV.lFileAdress, lMaxSize := MNPARAM_TEMPWRITECSVSIZE, lSize := _Intern.WriteCSV.lFileSize);

					FOR _i := 1 TO MNPARAM_CNT_CSVFILES DO

						IF _Intern.TOC.TocEntry[_i].xExist THEN

							_WriteToc(enable := TRUE, pMem := _Intern.WriteCSV.lFileAdress, lMaxSize := MNPARAM_TEMPWRITECSVSIZE, ContentRow := _Intern.TOC.TocEntry[_i] , lSize := _Intern.WriteCSV.lFileSize);

						END_IF

					END_FOR

					_WriteFileEnd(enable := TRUE, pMem := _Intern.WriteCSV.lFileAdress, lMaxSize := MNPARAM_TEMPWRITECSVSIZE, lSize := _Intern.WriteCSV.lFileSize);

					_TocExpState := tes_DeleteFileCSV;

					_sPathAndFilename := CONCAT(_Intern.ExpSettings.sPath, 'TOC.csv');

				//==============================================
				// Möglicherweise vorhandene Exportdatei löschen
				//==============================================
				tes_DeleteFileCSV:

					_deleteCSVFile(enable := TRUE, pDevice := ADR(_Intern.ExpSettings.sCfDeviceName), pName := ADR(_sPathAndFilename));

					IF _deleteCSVFile.status <> ERR_FUB_BUSY THEN

						_TocExpState := tes_CreateFileCSV;

					ELSE

						_xBusy := TRUE;

					END_IF

				//==============================================
				// Exportdatei erzeugen
				//==============================================
				tes_CreateFileCSV:

					_createCSVFile(enable := TRUE, pDevice := ADR(_Intern.ExpSettings.sCfDeviceName), pFile := ADR(_sPathAndFilename) );

					IF _createCSVFile.status = ERR_OK THEN

						_TocExpState := tes_WriteFileCSV;

					ELSIF _createCSVFile.status <> ERR_FUB_BUSY THEN

						_wIntStatus := MNPARAM_STAT_CREATECSV;
						_wIntAdStatus := _createCSVFile.status;

						_TocExpState := tes_FreeMemCSV;

						_Intern.Logger.logLevel 	:= arlogLEVEL_INFO;
						_Intern.Logger.text		:= 'FileCreate for Writing TOC File. Status : {##AttrVar2}';
						_Intern.Logger.var1		:= 0;
						_Intern.Logger.var2		:= _createCSVFile.status;

						_xFault := TRUE;

					ELSE

						_xBusy := TRUE;

					END_IF

				//==============================================
				// Exportdatei öffnen
				//==============================================
				tes_OpenFileCSV:

					_openCSVFile(enable := TRUE, pDevice := ADR(_Intern.ExpSettings.sCfDeviceName), pFile := ADR(_sPathAndFilename), mode := fiWRITE_ONLY);

					IF _openCSVFile.status = ERR_OK THEN

						_TocExpState := tes_WriteFileCSV;

					ELSIF _openCSVFile.status <> ERR_FUB_BUSY THEN

						_wIntStatus := MNPARAM_STAT_OPENCSV;
						_wIntAdStatus := _openCSVFile.status;

						_TocExpState := tes_FreeMemCSV;

						_Intern.Logger.logLevel := arlogLEVEL_INFO;
						_Intern.Logger.text		:= 'FileOpen for Writing TOC File. Status : {##AttrVar2}';
						_Intern.Logger.var1		:= 0;
						_Intern.Logger.var2		:= _openCSVFile.status;

						_xFault := TRUE;

					ELSE

						_xBusy := TRUE;

					END_IF

				//==============================================
				// Exportdatei schreiben
				//==============================================
				tes_WriteFileCSV:

					_writeCSVFile(enable := TRUE, ident := _createCSVFile.ident, offset := 0, pSrc :=_Intern.WriteCSV.lFileAdress, len := _Intern.WriteCSV.lFileSize);

					IF _writeCSVFile.status = ERR_OK THEN

						_TocExpState := tes_CloseFileCSV;

					ELSIF _writeCSVFile.status <> ERR_FUB_BUSY THEN

						_wIntStatus := MNPARAM_STAT_WRITECSV;
						_wIntAdStatus := _writeCSVFile.status;

						_TocExpState := tes_CloseFileCSV;

						_Intern.Logger.logLevel := arlogLEVEL_INFO;
						_Intern.Logger.text		:= 'FileWrite for Writing TOC File. Status : {##AttrVar2}';
						_Intern.Logger.var1		:= 0;
						_Intern.Logger.var2		:= _writeCSVFile.status;

						_xFault := TRUE;

					ELSE

						_xBusy := TRUE;

					END_IF

				//==============================================
				// Exportdatei schließen
				//==============================================
				tes_CloseFileCSV:

					_closeCSVFile(enable := TRUE, ident := _createCSVFile.ident);

					IF _closeCSVFile.status = ERR_OK THEN

						_TocExpState := tes_FreeMemCSV;

					ELSIF _closeCSVFile.status <> ERR_FUB_BUSY THEN

						IF NOT _xFault THEN

							_wIntStatus := MNPARAM_STAT_CLOSECSV;
							_wIntAdStatus := _closeCSVFile.status;

							_Intern.Logger.logLevel := arlogLEVEL_INFO;
							_Intern.Logger.text		:= 'FileClose for Writing TOC File. Status : {##AttrVar2}';
							_Intern.Logger.var1		:= 0;
							_Intern.Logger.var2		:= _closeCSVFile.status;

						END_IF

						_xFault := TRUE;

						_TocExpState := tes_FreeMemCSV;

					ELSE

						_xBusy := TRUE;

					END_IF

				//==============================================
				// Allokierten Speicher frei geben
				//==============================================
				tes_FreeMemCSV:

					_MemPartFree(enable := TRUE, ident  := _Intern.MemSettings.PartIdent, mem := _Intern.WriteCSV.lFileAdress);

					IF _MemPartFree.status = ERR_OK THEN

						_Intern.WriteCSV.lFileAdress := 0;
						_Intern.WriteCSV.lFileSize := 0;

						IF _xFault THEN

							Status := _wIntStatus;
							AdStatus := _wIntAdStatus;

							_TocExpState := tes_Log;

						ELSE

							Status := ERR_OK;
							AdStatus := 0;

							_xReady := TRUE;

							_TocExpState := tes_AllocMemCSV;

						END_IF

					ELSIF _MemPartFree.status <> ERR_FUB_BUSY THEN

						_Intern.WriteCSV.lFileAdress := 0;
						_Intern.WriteCSV.lFileSize := 0;

						IF _xFault THEN

							Status := _wIntStatus;
							AdStatus := _wIntAdStatus;

						ELSE

							Status := MNPARAM_STAT_EXPFREEMEM;
							AdStatus := _MemPartFree.status;

							_Intern.Logger.logLevel := arlogLEVEL_INFO;
							_Intern.Logger.text		:= 'FreeMem for Writing TOC File. Status : {##AttrVar2}';
							_Intern.Logger.var1		:= 0;
							_Intern.Logger.var2		:= _MemPartFree.status;

						END_IF

						_TocExpState := tes_Log;

					ELSE

						_xBusy := TRUE;

					END_IF

				//==============
				// Fehler loggen
				//==============
				tes_Log:

					_Intern.Logger();

					IF _Intern.Logger.status <> ERR_FUB_BUSY THEN

						Status := _wIntStatus;
						AdStatus := _wIntAdStatus;

						_TocExpState := tes_AllocMemCSV;

						_xReady := TRUE;

					ELSE

						_xBusy := TRUE;

					END_IF

			END_CASE

			UNTIL

			_xBusy OR _xReady

		END_REPEAT

		IF _xBusy THEN
			Status := ERR_FUB_BUSY;
		END_IF

	ELSE

		_TocExpState := tes_AllocMemCSV;

		Status := ERR_FUB_ENABLE_FALSE;
		AdStatus := 0;

	END_IF

END_FUNCTION_BLOCK
```

#### _DefActContainer.st - Fülle ActContainer
```iecst
(********************************************************************
 * COPYRIGHT -- Herbert Kannegiesser GmbH
 ********************************************************************
 * Program: mnParam
 * File: _DefActContainer.st
 * Author: hunholz
 * Created: February 17, 2012
 ********************************************************************
 * Implementation of program mnParam
 ********************************************************************)

(* Fülle ActContainer *)
FUNCTION_BLOCK _DefActContainer

	IF Enable THEN

		Status := ERR_OK;

		//=======================
		// Auf Nullpointer prüfen
		//=======================

		IF pIntern = 0 THEN
			Status := MNPARAM_STAT_NULLPOINTER;
			RETURN;
		END_IF

		_Intern ACCESS pIntern;

		IF _Intern.DataObjects.Adress.lContainer = 0 THEN
			Status := MNPARAM_STAT_NULLPOINTER;
			RETURN;
		END_IF

		_DoContainer ACCESS _Intern.DataObjects.Adress.lContainer;

		// Containerindex zulässig ?
		IF bContainerIdx > _Intern.DataObjects.MaxIndex.lContainer THEN

			Status := MNPARAM_STAT_CONTAINER_NOT_VALID;

			RETURN;

		END_IF

		// Datenobjekt- und Dateinamen ok?

		IF (brsstrcmp(ADR(_DoContainer.Container[bContainerIdx].sNameDataObj), ADR('')) = 0) OR (brsstrcmp(ADR(_DoContainer.Container[bContainerIdx].sNameCsv), ADR('')) = 0) THEN

			Status := MNPARAM_STAT_CONTAINER_NOT_VALID;

			RETURN;

		END_IF

		// Ist die Rootvariable bei indirekter Parametrierung OK ?

		IF _DoContainer.Container[bContainerIdx].bDirectParam = 0 AND (PV_xgetadr(ADR(_DoContainer.Container[bContainerIdx].sStrucRoot), ADR(_lPVadress), ADR(_lPVlen)) <> ERR_OK) THEN

			Status := MNPARAM_STAT_CONTAINER_NOT_VALID;

			RETURN;

		END_IF

		_Intern.ActContainer.siContainerID := _DoContainer.Container[bContainerIdx].siContainerID;

		_Intern.ActContainer.bDirect := _DoContainer.Container[bContainerIdx].bDirectParam;

		_Intern.ActContainer.wMinBound := _DoContainer.Container[bContainerIdx].wMinBound;
		_Intern.ActContainer.wDimension := _DoContainer.Container[bContainerIdx].wDimension;

		IF wInstanceIdx < _Intern.ActContainer.wMinBound THEN

			Status := MNPARAM_STAT_CONTINST_NOT_VALID;

			RETURN;

		END_IF

		IF _Intern.ActContainer.wDimension <= 1 AND wInstanceIdx > _Intern.ActContainer.wMinBound THEN

			Status := MNPARAM_STAT_CONTINST_NOT_VALID;

			RETURN;

		END_IF

		IF wInstanceIdx > (_Intern.ActContainer.wMinBound + _Intern.ActContainer.wDimension - 1) THEN

			Status := MNPARAM_STAT_CONTINST_NOT_VALID;

			RETURN;

		END_IF

		_Intern.ActContainer.wIndexIndirect := wInstanceIdx;

		IF _DoContainer.Container[bContainerIdx].bDirectParam = 0 THEN

			// Indirekte Parametrierung

			_wDimension := MAX(1,_Intern.ActContainer.wDimension);

			_Intern.ActContainer.lAdressStructRoot := _lPVadress;
			_Intern.ActContainer.lSizeStructRoot := _lPVlen;

			_Intern.ActContainer.sDoNameDef := CONCAT(_DoContainer.Container[bContainerIdx].sNameDataObj,'d');
			_Intern.ActContainer.sDoNameDefNum := CONCAT(_DoContainer.Container[bContainerIdx].sNameDataObj, 'Nd');
			_Intern.ActContainer.sDoNameDefString := CONCAT(_DoContainer.Container[bContainerIdx].sNameDataObj, 'Sd');
			_Intern.ActContainer.sStrucRoot := _DoContainer.Container[bContainerIdx].sStrucRoot;

			_Intern.ActContainer.sIndex := '';
			IF (_Intern.ActContainer.wMinBound + _wDimension - 1) > 9999 AND  _Intern.ActContainer.wIndexIndirect  < 10000 THEN
				_Intern.ActContainer.sIndex := CONCAT(_Intern.ActContainer.sIndex,'0');
			END_IF
			IF (_Intern.ActContainer.wMinBound + _wDimension - 1) > 999 AND  _Intern.ActContainer.wIndexIndirect  < 1000 THEN
				_Intern.ActContainer.sIndex := CONCAT(_Intern.ActContainer.sIndex,'0');
			END_IF
			IF (_Intern.ActContainer.wMinBound + _wDimension - 1) > 99 AND  _Intern.ActContainer.wIndexIndirect  < 100 THEN
				_Intern.ActContainer.sIndex := CONCAT(_Intern.ActContainer.sIndex,'0');
			END_IF
			IF (_Intern.ActContainer.wMinBound + _wDimension - 1) > 9 AND  _Intern.ActContainer.wIndexIndirect  < 10 THEN
				_Intern.ActContainer.sIndex := CONCAT(_Intern.ActContainer.sIndex,'0');
			END_IF

			_sIndex := UINT_TO_STRING(_Intern.ActContainer.wIndexIndirect);
			_Intern.ActContainer.sIndex := CONCAT(_Intern.ActContainer.sIndex,_sIndex);

			_Intern.ActContainer.sDoName := CONCAT(_DoContainer.Container[bContainerIdx].sNameDataObj, _Intern.ActContainer.sIndex);

			_Intern.ActContainer.sDoNameNum := CONCAT(_DoContainer.Container[bContainerIdx].sNameDataObj, _Intern.ActContainer.sIndex);
			_Intern.ActContainer.sDoNameNum := CONCAT(_Intern.ActContainer.sDoNameNum, 'N');

			_Intern.ActContainer.sDoNameString := CONCAT(_DoContainer.Container[bContainerIdx].sNameDataObj, _Intern.ActContainer.sIndex);
			_Intern.ActContainer.sDoNameString := CONCAT(_Intern.ActContainer.sDoNameString, 'S');

			_Intern.ActContainer.sCsvName := CONCAT(_DoContainer.Container[bContainerIdx].sNameCsv, _Intern.ActContainer.sIndex);
			_Intern.ActContainer.sCsvName := CONCAT(_Intern.ActContainer.sCsvName, MNPARAM_FILESUFF);

		ELSE

			// Direkte Parametrierung

			_Intern.ActContainer.lAdressStructRoot := 0;
			_Intern.ActContainer.lSizeStructRoot := 0;

			_Intern.ActContainer.sDoName := '';
			_Intern.ActContainer.sDoNameDef := '';
			_Intern.ActContainer.sDoNameDefNum := '';
			_Intern.ActContainer.sDoNameDefString := '';
			_Intern.ActContainer.sStrucRoot := '';

			_Intern.ActContainer.sDoNameNum := CONCAT(_DoContainer.Container[bContainerIdx].sNameDataObj, 'N');
			_Intern.ActContainer.sDoNameString := CONCAT(_DoContainer.Container[bContainerIdx].sNameDataObj, 'S');

			_Intern.ActContainer.sCsvName := CONCAT(_DoContainer.Container[bContainerIdx].sNameCsv, MNPARAM_FILESUFF);

		END_IF

		_Intern.ActContainer.lCountParamNum := _DoContainer.Container[bContainerIdx].lCountNum;
		_Intern.ActContainer.lCountParamString := _DoContainer.Container[bContainerIdx].lCountString;

	ELSE

		Status := ERR_FUB_ENABLE_FALSE;

	END_IF

END_FUNCTION_BLOCK
```
